LIN {X 0,Y 242.041,Z 125.949,A -85,B 0,C 180,E1 -19236.009,E2 -19236.009} C_VEL
LIN {X 0,Y 242.05,Z 125.947,A -85,B 0,C 180,E1 -19239.604,E2 -19239.604} C_VEL
LIN {X 0,Y 242.178,Z 125.932,A -85,B 0,C 180,E1 -19243.274,E2 -19243.274} C_VEL
LIN {X 0,Y 242.183,Z 125.929,A -85,B 0,C 180,E1 -19248.274,E2 -19248.274} C_VEL
LIN {X 0,Y 242.383,Z 125.908,A -85,B 0,C 180,E1 -19251.659,E2 -19251.659} C_VEL
LIN {X 0,Y 242.244,Z 125.935,A -85,B 0,C 180,E1 -19255.002,E2 -19255.002} C_VEL
LIN {X 0,Y 242.634,Z 125.882,A -85,B 0,C 180,E1 -19258.335,E2 -19258.335} C_VEL
LIN {X 0,Y 242.641,Z 125.873,A -85,B 0,C 180,E1 -19261.654,E2 -19261.654} C_VEL
LIN {X 0,Y 242.413,Z 125.908,A -85,B 0,C 180,E1 -19266.654,E2 -19266.654} C_VEL
LIN {X 0,Y 242.272,Z 125.921,A -85,B 0,C 180,E1 -19270.018,E2 -19270.018} C_VEL
LIN {X 0,Y 242.169,Z 125.946,A -85,B 0,C 180,E1 -19275.134,E2 -19275.134} C_VEL
LIN {X 0,Y 242.074,Z 125.958,A -85,B 0,C 180,E1 -19278.618,E2 -19278.618} C_VEL
LIN {X 0,Y 242.029,Z 126.021,A -85,B 0,C 180,E1 -19282.565,E2 -19282.565} C_VEL
LIN {X 0,Y 242.806,Z 128.403,A -85,B 0,C 180,E1 -19282.995,E2 -19282.995} C_VEL
LIN {X 0,Y 244.693,Z 130.652,A -85,B 0,C 180,E1 -19283.815,E2 -19283.815} C_VEL
LIN {X 0,Y 246.169,Z 131.607,A -85,B 0,C 180,E1 -19284.391,E2 -19284.391} C_VEL
LIN {X 0,Y 247.934,Z 134.724,A -85,B 0,C 180,E1 -19285.156,E2 -19285.156} C_VEL
LIN {X 0,Y 250.263,Z 137.17,A -85,B 0,C 180,E1 -19286.045,E2 -19286.045} C_VEL
LIN {X 0,Y 252.842,Z 140.696,A -85,B 0,C 180,E1 -19287.026,E2 -19287.026} C_VEL
LIN {X 0,Y 254.234,Z 142.51,A -85,B 0,C 180,E1 -19287.534,E2 -19287.534} C_VEL
LIN {X 0,Y 258.183,Z 148.167,A -85,B 0,C 180,E1 -19288.938,E2 -19288.938} C_VEL
LIN {X 0,Y 265.416,Z 159.264,A -85,B 0,C 180,E1 -19291.315,E2 -19291.315} C_VEL
LIN {X 0,Y 272.928,Z 172.626,A -85,B 0,C 180,E1 -19293.606,E2 -19293.606} C_VEL
LIN {X 0,Y 279.601,Z 186.169,A -85,B 0,C 180,E1 -19295.519,E2 -19295.519} C_VEL
LIN {X 0,Y 280.351,Z 187.777,A -85,B 0,C 180,E1 -19295.727,E2 -19295.727} C_VEL
LIN {X 0,Y 276.357,Z 261.18,A -85,B 0,C 180,E1 -19297.607,E2 -19297.607} C_VEL
LIN {X 0,Y 274.792,Z 275.361,A -85,B 0,C 180,E1 -19298.216,E2 -19298.216} C_VEL
LIN {X 0,Y 272.705,Z 288.841,A -85,B 0,C 180,E1 -19299.068,E2 -19299.068} C_VEL
LIN {X 0,Y 270.18,Z 301.704,A -85,B 0,C 180,E1 -19300.169,E2 -19300.169} C_VEL
LIN {X 0,Y 267.285,Z 313.739,A -85,B 0,C 180,E1 -19301.491,E2 -19301.491} C_VEL
LIN {X 0,Y 263.786,Z 325.88,A -85,B 0,C 180,E1 -19303.166,E2 -19303.166} C_VEL
LIN {X 0,Y 260.3,Z 336.639,A -85,B 0,C 180,E1 -19305.032,E2 -19305.032} C_VEL
LIN {X 0,Y 256.62,Z 346.76,A -85,B 0,C 180,E1 -19307.207,E2 -19307.207} C_VEL
LIN {X 0,Y 252.911,Z 356.201,A -85,B 0,C 180,E1 -19309.751,E2 -19309.751} C_VEL
LIN {X 0,Y 249.787,Z 363.635,A -85,B 0,C 180,E1 -19312.266,E2 -19312.266} C_VEL
LIN {X 0,Y 246.665,Z 370.6,A -85,B 0,C 180,E1 -19315.258,E2 -19315.258} C_VEL
LIN {X 0,Y 244.554,Z 375.362,A -85,B 0,C 180,E1 -19317.88,E2 -19317.88} C_VEL
LIN {X 0,Y 242.846,Z 379.053,A -85,B 0,C 180,E1 -19320.526,E2 -19320.526} C_VEL
LIN {X 0,Y 241.181,Z 382.568,A -85,B 0,C 180,E1 -19324.079,E2 -19324.079} C_VEL
LIN {X 0,Y 240.608,Z 383.728,A -85,B 0,C 180,E1 -19325.86,E2 -19325.86} C_VEL
LIN {X 0,Y 239.858,Z 384.91,A -85,B 0,C 180,E1 -19329.412,E2 -19329.412} C_VEL
LIN {X 0,Y 239.521,Z 384.657,A -85,B 0,C 180,E1 -19332.935,E2 -19332.935} C_VEL
LIN {X 0,Y 239.567,Z 382.993,A -85,B 0,C 180,E1 -19336.424,E2 -19336.424} C_VEL
LIN {X 0,Y 239.857,Z 379.919,A -85,B 0,C 180,E1 -19339.872,E2 -19339.872} C_VEL
LIN {X 0,Y 240.373,Z 376.626,A -85,B 0,C 180,E1 -19342.437,E2 -19342.437} C_VEL
LIN {X 0,Y 240.994,Z 372.483,A -85,B 0,C 180,E1 -19344.979,E2 -19344.979} C_VEL
LIN {X 0,Y 241.907,Z 367.319,A -85,B 0,C 180,E1 -19347.5,E2 -19347.5} C_VEL
LIN {X 0,Y 243.405,Z 359.946,A -85,B 0,C 180,E1 -19350.411,E2 -19350.411} C_VEL
LIN {X 0,Y 245.384,Z 350.779,A -85,B 0,C 180,E1 -19353.281,E2 -19353.281} C_VEL
LIN {X 0,Y 247.431,Z 341.232,A -85,B 0,C 180,E1 -19355.692,E2 -19355.692} C_VEL
LIN {X 0,Y 249.463,Z 330.6,A -85,B 0,C 180,E1 -19357.892,E2 -19357.892} C_VEL
LIN {X 0,Y 251.81,Z 318.828,A -85,B 0,C 180,E1 -19359.841,E2 -19359.841} C_VEL
LIN {X 0,Y 254.053,Z 305.76,A -85,B 0,C 180,E1 -19361.567,E2 -19361.567} C_VEL
LIN {X 0,Y 255.854,Z 292.944,A -85,B 0,C 180,E1 -19362.894,E2 -19362.894} C_VEL
LIN {X 0,Y 257.346,Z 279.852,A -85,B 0,C 180,E1 -19363.923,E2 -19363.923} C_VEL
LIN {X 0,Y 258.5,Z 265.758,A -85,B 0,C 180,E1 -19364.714,E2 -19364.714} C_VEL
LIN {X 0,Y 259.312,Z 249.37,A -85,B 0,C 180,E1 -19365.27,E2 -19365.27} C_VEL
LIN {X 0,Y 262.369,Z 171.816,A -85,B 0,C 180,E1 -19367.319,E2 -19367.319} C_VEL
LIN {X 0,Y 253.658,Z 149.318,A -85,B 0,C 180,E1 -19369.1,E2 -19369.1} C_VEL
LIN {X 0,Y 248.74,Z 138.889,A -85,B 0,C 180,E1 -19370.096,E2 -19370.096} C_VEL
LIN {X 0,Y 243.439,Z 129.314,A -85,B 0,C 180,E1 -19371.164,E2 -19371.164} C_VEL
LIN {X 0,Y 242.187,Z 126.552,A -85,B 0,C 180,E1 -19371.442,E2 -19371.442} C_VEL
LIN {X 0,Y 242.072,Z 125.958,A -85,B 0,C 180,E1 -19371.532,E2 -19371.532} C_VEL
LIN {X 0,Y 242.035,Z 125.96,A -85,B 0,C 180,E1 -19375.839,E2 -19375.839} C_VEL
LIN {X 0,Y 241.999,Z 125.965,A -85,B 0,C 180,E1 -19379.581,E2 -19379.581} C_VEL
LIN {X 0,Y 241.961,Z 125.971,A -85,B 0,C 180,E1 -19383.493,E2 -19383.493} C_VEL
LIN {X 0,Y 242.004,Z 125.964,A -85,B 0,C 180,E1 -19387.576,E2 -19387.576} C_VEL
LIN {X 0,Y 242.025,Z 125.957,A -85,B 0,C 180,E1 -19391.9,E2 -19391.9} C_VEL
LIN {X 0,Y 241.997,Z 125.962,A -85,B 0,C 180,E1 -19396.552,E2 -19396.552} C_VEL
LIN {X 0,Y 241.984,Z 125.953,A -85,B 0,C 180,E1 -19400.295,E2 -19400.295} C_VEL
LIN {X 0,Y 242.012,Z 125.957,A -85,B 0,C 180,E1 -19404.501,E2 -19404.501} C_VEL
LIN {X 0,Y 241.951,Z 125.964,A -85,B 0,C 180,E1 -19408.484,E2 -19408.484} C_VEL
LIN {X 0,Y 241.982,Z 125.944,A -85,B 0,C 180,E1 -19412.317,E2 -19412.317} C_VEL
LIN {X 0,Y 242.062,Z 125.957,A -85,B 0,C 180,E1 -19416.023,E2 -19416.023} C_VEL
LIN {X 0,Y 242.068,Z 125.952,A -85,B 0,C 180,E1 -19419.617,E2 -19419.617} C_VEL
LIN {X 0,Y 242.146,Z 125.946,A -85,B 0,C 180,E1 -19423.283,E2 -19423.283} C_VEL
LIN {X 0,Y 242.172,Z 125.942,A -85,B 0,C 180,E1 -19428.285,E2 -19428.285} C_VEL
LIN {X 0,Y 242.421,Z 125.897,A -85,B 0,C 180,E1 -19431.671,E2 -19431.671} C_VEL
LIN {X 0,Y 242.251,Z 125.913,A -85,B 0,C 180,E1 -19435.013,E2 -19435.013} C_VEL
LIN {X 0,Y 242.629,Z 125.884,A -85,B 0,C 180,E1 -19438.346,E2 -19438.346} C_VEL
LIN {X 0,Y 242.628,Z 125.879,A -85,B 0,C 180,E1 -19441.665,E2 -19441.665} C_VEL
LIN {X 0,Y 242.253,Z 125.909,A -85,B 0,C 180,E1 -19444.875,E2 -19444.875} C_VEL
LIN {X 0,Y 241.585,Z 126.003,A -85,B 0,C 180,E1 -19446.265,E2 -19446.265} C_VEL
LIN {X 0,Y 238.754,Z 126.366,A -85,B 0,C 180,E1 -19448.532,E2 -19448.532} C_VEL
LIN {X 0,Y 235.487,Z 126.773,A -85,B 0,C 180,E1 -19451.328,E2 -19451.328} C_VEL
LIN {X 0,Y 235.124,Z 126.815,A -85,B 0,C 180,E1 -19452.297,E2 -19452.297} C_VEL
LIN {X 0,Y 235.092,Z 126.822,A -85,B 0,C 180,E1 -19456.946,E2 -19456.946} C_VEL
LIN {X 0,Y 234.991,Z 126.837,A -85,B 0,C 180,E1 -19462.015,E2 -19462.015} C_VEL
LIN {X 0,Y 234.969,Z 126.835,A -85,B 0,C 180,E1 -19466.663,E2 -19466.663} C_VEL
LIN {X 0,Y 234.932,Z 126.843,A -85,B 0,C 180,E1 -19470.573,E2 -19470.573} C_VEL
LIN {X 0,Y 234.932,Z 126.844,A -85,B 0,C 180,E1 -19474.643,E2 -19474.643} C_VEL
LIN {X 0,Y 234.916,Z 126.844,A -85,B 0,C 180,E1 -19478.941,E2 -19478.941} C_VEL
LIN {X 0,Y 234.882,Z 126.853,A -85,B 0,C 180,E1 -19483.493,E2 -19483.493} C_VEL
LIN {X 0,Y 234.883,Z 126.853,A -85,B 0,C 180,E1 -19486.517,E2 -19486.517} C_VEL
LIN {X 0,Y 234.919,Z 127.017,A -85,B 0,C 180,E1 -19488.637,E2 -19488.637} C_VEL
LIN {X 0,Y 236.99,Z 134.697,A -85,B 0,C 180,E1 -19491.697,E2 -19491.697} C_VEL
LIN {X 0,Y 243.013,Z 147.893,A -85,B 0,C 180,E1 -19493.045,E2 -19493.045} C_VEL
LIN {X 0,Y 251.14,Z 167.812,A -85,B 0,C 180,E1 -19494.814,E2 -19494.814} C_VEL
LIN {X 0,Y 253.217,Z 173.701,A -85,B 0,C 180,E1 -19495.269,E2 -19495.269} C_VEL
LIN {X 0,Y 255.518,Z 191.759,A -85,B 0,C 180,E1 -19496.129,E2 -19496.129} C_VEL
LIN {X 0,Y 252.428,Z 272.237,A -85,B 0,C 180,E1 -19498.359,E2 -19498.359} C_VEL
LIN {X 0,Y 251.193,Z 286.32,A -85,B 0,C 180,E1 -19499.007,E2 -19499.007} C_VEL
LIN {X 0,Y 249.679,Z 299.519,A -85,B 0,C 180,E1 -19499.911,E2 -19499.911} C_VEL
LIN {X 0,Y 247.651,Z 313.005,A -85,B 0,C 180,E1 -19501.158,E2 -19501.158} C_VEL
LIN {X 0,Y 245.502,Z 326.007,A -85,B 0,C 180,E1 -19502.743,E2 -19502.743} C_VEL
LIN {X 0,Y 243.137,Z 337.78,A -85,B 0,C 180,E1 -19504.537,E2 -19504.537} C_VEL
LIN {X 0,Y 241.554,Z 345.588,A -85,B 0,C 180,E1 -19505.966,E2 -19505.966} C_VEL
LIN {X 0,Y 239.418,Z 355.067,A -85,B 0,C 180,E1 -19508.024,E2 -19508.024} C_VEL
LIN {X 0,Y 237.365,Z 364.58,A -85,B 0,C 180,E1 -19510.546,E2 -19510.546} C_VEL
LIN {X 0,Y 235.614,Z 373.622,A -85,B 0,C 180,E1 -19513.541,E2 -19513.541} C_VEL
LIN {X 0,Y 234.356,Z 379.977,A -85,B 0,C 180,E1 -19516.121,E2 -19516.121} C_VEL
LIN {X 0,Y 233.464,Z 385.192,A -85,B 0,C 180,E1 -19518.719,E2 -19518.719} C_VEL
LIN {X 0,Y 233,Z 389.396,A -85,B 0,C 180,E1 -19521.328,E2 -19521.328} C_VEL
LIN {X 0,Y 232.741,Z 393.621,A -85,B 0,C 180,E1 -19524.805,E2 -19524.805} C_VEL
LIN {X 0,Y 232.76,Z 396.365,A -85,B 0,C 180,E1 -19528.272,E2 -19528.272} C_VEL
LIN {X 0,Y 232.83,Z 397.21,A -85,B 0,C 180,E1 -19530.002,E2 -19530.002} C_VEL
LIN {X 0,Y 232.667,Z 397.873,A -85,B 0,C 180,E1 -19533.466,E2 -19533.466} C_VEL
LIN {X 0,Y 232.829,Z 397.211,A -85,B 0,C 180,E1 -19536.937,E2 -19536.937} C_VEL
LIN {X 0,Y 233.482,Z 395.231,A -85,B 0,C 180,E1 -19540.407,E2 -19540.407} C_VEL
LIN {X 0,Y 234.709,Z 391.888,A -85,B 0,C 180,E1 -19543.862,E2 -19543.862} C_VEL
LIN {X 0,Y 236.804,Z 387.097,A -85,B 0,C 180,E1 -19547.267,E2 -19547.267} C_VEL
LIN {X 0,Y 239.552,Z 380.722,A -85,B 0,C 180,E1 -19550.616,E2 -19550.616} C_VEL
LIN {X 0,Y 242.692,Z 373.665,A -85,B 0,C 180,E1 -19553.467,E2 -19553.467} C_VEL
LIN {X 0,Y 245.851,Z 366.318,A -85,B 0,C 180,E1 -19555.848,E2 -19555.848} C_VEL
LIN {X 0,Y 249.475,Z 357.524,A -85,B 0,C 180,E1 -19558.158,E2 -19558.158} C_VEL
LIN {X 0,Y 253.373,Z 347.313,A -85,B 0,C 180,E1 -19560.318,E2 -19560.318} C_VEL
LIN {X 0,Y 256.969,Z 336.685,A -85,B 0,C 180,E1 -19562.14,E2 -19562.14} C_VEL
LIN {X 0,Y 260.744,Z 324.554,A -85,B 0,C 180,E1 -19563.776,E2 -19563.776} C_VEL
LIN {X 0,Y 263.987,Z 311.763,A -85,B 0,C 180,E1 -19565.152,E2 -19565.152} C_VEL
LIN {X 0,Y 266.924,Z 298.45,A -85,B 0,C 180,E1 -19566.214,E2 -19566.214} C_VEL
LIN {X 0,Y 269.32,Z 283.857,A -85,B 0,C 180,E1 -19567.059,E2 -19567.059} C_VEL
LIN {X 0,Y 270.863,Z 269.38,A -85,B 0,C 180,E1 -19567.616,E2 -19567.616} C_VEL
LIN {X 0,Y 274.782,Z 197.77,A -85,B 0,C 180,E1 -19569.471,E2 -19569.471} C_VEL
LIN {X 0,Y 268.635,Z 183.99,A -85,B 0,C 180,E1 -19571.343,E2 -19571.343} C_VEL
LIN {X 0,Y 262.523,Z 172.024,A -85,B 0,C 180,E1 -19573.303,E2 -19573.303} C_VEL
LIN {X 0,Y 257.036,Z 162.531,A -85,B 0,C 180,E1 -19575.163,E2 -19575.163} C_VEL
LIN {X 0,Y 252.081,Z 154.456,A -85,B 0,C 180,E1 -19576.971,E2 -19576.971} C_VEL
LIN {X 0,Y 248.527,Z 149.046,A -85,B 0,C 180,E1 -19578.348,E2 -19578.348} C_VEL
LIN {X 0,Y 244.891,Z 143.679,A -85,B 0,C 180,E1 -19579.843,E2 -19579.843} C_VEL
LIN {X 0,Y 241.577,Z 138.818,A -85,B 0,C 180,E1 -19581.309,E2 -19581.309} C_VEL
LIN {X 0,Y 237.543,Z 133.584,A -85,B 0,C 180,E1 -19583.203,E2 -19583.203} C_VEL
LIN {X 0,Y 236.83,Z 132.267,A -85,B 0,C 180,E1 -19583.588,E2 -19583.588} C_VEL
LIN {X 0,Y 235.994,Z 129.663,A -85,B 0,C 180,E1 -19585.535,E2 -19585.535} C_VEL
LIN {X 0,Y 234.948,Z 126.839,A -85,B 0,C 180,E1 -19587.925,E2 -19587.925} C_VEL
LIN {X 0,Y 234.918,Z 126.842,A -85,B 0,C 180,E1 -19591.396,E2 -19591.396} C_VEL
LIN {X 0,Y 234.97,Z 126.832,A -85,B 0,C 180,E1 -19595.239,E2 -19595.239} C_VEL
LIN {X 0,Y 235.013,Z 126.827,A -85,B 0,C 180,E1 -19598.965,E2 -19598.965} C_VEL
LIN {X 0,Y 235.111,Z 126.814,A -85,B 0,C 180,E1 -19603.056,E2 -19603.056} C_VEL
LIN {X 0,Y 235.116,Z 126.81,A -85,B 0,C 180,E1 -19607.917,E2 -19607.917} C_VEL
LIN {X 0,Y 235.323,Z 126.789,A -85,B 0,C 180,E1 -19611.407,E2 -19611.407} C_VEL
LIN {X 0,Y 235.36,Z 126.78,A -85,B 0,C 180,E1 -19613.135,E2 -19613.135} C_VEL
LIN {X 0,Y 235.593,Z 126.758,A -85,B 0,C 180,E1 -19618.285,E2 -19618.285} C_VEL
LIN {X 0,Y 235.6,Z 126.749,A -85,B 0,C 180,E1 -19621.704,E2 -19621.704} C_VEL
LIN {X 0,Y 235.364,Z 126.788,A -85,B 0,C 180,E1 -19626.854,E2 -19626.854} C_VEL
LIN {X 0,Y 235.219,Z 126.802,A -85,B 0,C 180,E1 -19630.321,E2 -19630.321} C_VEL
LIN {X 0,Y 235.116,Z 126.82,A -85,B 0,C 180,E1 -19635.6,E2 -19635.6} C_VEL
LIN {X 0,Y 234.996,Z 126.84,A -85,B 0,C 180,E1 -19639.711,E2 -19639.711} C_VEL
LIN {X 0,Y 235.78,Z 129.313,A -85,B 0,C 180,E1 -19640.21,E2 -19640.21} C_VEL
LIN {X 0,Y 237.696,Z 131.568,A -85,B 0,C 180,E1 -19641.16,E2 -19641.16} C_VEL
LIN {X 0,Y 239.366,Z 132.759,A -85,B 0,C 180,E1 -19641.909,E2 -19641.909} C_VEL
LIN {X 0,Y 241.227,Z 135.882,A -85,B 0,C 180,E1 -19642.814,E2 -19642.814} C_VEL
LIN {X 0,Y 243.587,Z 138.113,A -85,B 0,C 180,E1 -19643.817,E2 -19643.817} C_VEL
LIN {X 0,Y 245.898,Z 141.51,A -85,B 0,C 180,E1 -19644.814,E2 -19644.814} C_VEL
LIN {X 0,Y 247.465,Z 143.234,A -85,B 0,C 180,E1 -19645.432,E2 -19645.432} C_VEL
LIN {X 0,Y 251.784,Z 149.168,A -85,B 0,C 180,E1 -19647.107,E2 -19647.107} C_VEL
LIN {X 0,Y 254.835,Z 153.563,A -85,B 0,C 180,E1 -19648.228,E2 -19648.228} C_VEL
LIN {X 0,Y 261.686,Z 164.264,A -85,B 0,C 180,E1 -19650.577,E2 -19650.577} C_VEL
LIN {X 0,Y 269.258,Z 178.011,A -85,B 0,C 180,E1 -19652.987,E2 -19652.987} C_VEL
LIN {X 0,Y 275.138,Z 190.241,A -85,B 0,C 180,E1 -19654.746,E2 -19654.746} C_VEL
LIN {X 0,Y 271.184,Z 261.131,A -85,B 0,C 180,E1 -19656.594,E2 -19656.594} C_VEL
LIN {X 0,Y 269.572,Z 275.306,A -85,B 0,C 180,E1 -19657.204,E2 -19657.204} C_VEL
LIN {X 0,Y 267.324,Z 289.177,A -85,B 0,C 180,E1 -19658.085,E2 -19658.085} C_VEL
LIN {X 0,Y 264.919,Z 301.058,A -85,B 0,C 180,E1 -19659.104,E2 -19659.104} C_VEL
LIN {X 0,Y 261.708,Z 313.991,A -85,B 0,C 180,E1 -19660.535,E2 -19660.535} C_VEL
LIN {X 0,Y 258.28,Z 325.511,A -85,B 0,C 180,E1 -19662.138,E2 -19662.138} C_VEL
LIN {X 0,Y 254.461,Z 336.758,A -85,B 0,C 180,E1 -19664.099,E2 -19664.099} C_VEL
LIN {X 0,Y 250.95,Z 346.031,A -85,B 0,C 180,E1 -19666.105,E2 -19666.105} C_VEL
LIN {X 0,Y 247.131,Z 355.357,A -85,B 0,C 180,E1 -19668.606,E2 -19668.606} C_VEL
LIN {X 0,Y 243.936,Z 362.668,A -85,B 0,C 180,E1 -19671.057,E2 -19671.057} C_VEL
LIN {X 0,Y 241.337,Z 368.256,A -85,B 0,C 180,E1 -19673.343,E2 -19673.343} C_VEL
LIN {X 0,Y 238.836,Z 373.518,A -85,B 0,C 180,E1 -19676.004,E2 -19676.004} C_VEL
LIN {X 0,Y 236.823,Z 377.698,A -85,B 0,C 180,E1 -19678.711,E2 -19678.711} C_VEL
LIN {X 0,Y 235.202,Z 380.863,A -85,B 0,C 180,E1 -19681.437,E2 -19681.437} C_VEL
LIN {X 0,Y 233.73,Z 383.725,A -85,B 0,C 180,E1 -19685.102,E2 -19685.102} C_VEL
LIN {X 0,Y 232.848,Z 385.078,A -85,B 0,C 180,E1 -19688.763,E2 -19688.763} C_VEL
LIN {X 0,Y 232.438,Z 384.953,A -85,B 0,C 180,E1 -19692.398,E2 -19692.398} C_VEL
LIN {X 0,Y 232.461,Z 383.408,A -85,B 0,C 180,E1 -19696.001,E2 -19696.001} C_VEL
LIN {X 0,Y 232.714,Z 380.456,A -85,B 0,C 180,E1 -19699.558,E2 -19699.558} C_VEL
LIN {X 0,Y 233.214,Z 377.292,A -85,B 0,C 180,E1 -19702.204,E2 -19702.204} C_VEL
LIN {X 0,Y 233.861,Z 373.229,A -85,B 0,C 180,E1 -19704.825,E2 -19704.825} C_VEL
LIN {X 0,Y 234.763,Z 368.191,A -85,B 0,C 180,E1 -19707.424,E2 -19707.424} C_VEL
LIN {X 0,Y 236.274,Z 360.973,A -85,B 0,C 180,E1 -19710.424,E2 -19710.424} C_VEL
LIN {X 0,Y 237.939,Z 353.421,A -85,B 0,C 180,E1 -19712.96,E2 -19712.96} C_VEL
LIN {X 0,Y 240.041,Z 344.038,A -85,B 0,C 180,E1 -19715.538,E2 -19715.538} C_VEL
LIN {X 0,Y 242.243,Z 333.398,A -85,B 0,C 180,E1 -19717.919,E2 -19717.919} C_VEL
LIN {X 0,Y 244.585,Z 322.217,A -85,B 0,C 180,E1 -19719.925,E2 -19719.925} C_VEL
LIN {X 0,Y 246.849,Z 309.877,A -85,B 0,C 180,E1 -19721.702,E2 -19721.702} C_VEL
LIN {X 0,Y 248.676,Z 298.056,A -85,B 0,C 180,E1 -19723.065,E2 -19723.065} C_VEL
LIN {X 0,Y 250.381,Z 285.154,A -85,B 0,C 180,E1 -19724.215,E2 -19724.215} C_VEL
LIN {X 0,Y 251.769,Z 270.528,A -85,B 0,C 180,E1 -19725.168,E2 -19725.168} C_VEL
LIN {X 0,Y 252.65,Z 255.97,A -85,B 0,C 180,E1 -19725.786,E2 -19725.786} C_VEL
LIN {X 0,Y 256.09,Z 173.861,A -85,B 0,C 180,E1 -19728.003,E2 -19728.003} C_VEL
LIN {X 0,Y 249.273,Z 155.648,A -85,B 0,C 180,E1 -19729.466,E2 -19729.466} C_VEL
LIN {X 0,Y 243.752,Z 143.416,A -85,B 0,C 180,E1 -19730.634,E2 -19730.634} C_VEL
LIN {X 0,Y 236.457,Z 130.343,A -85,B 0,C 180,E1 -19732.171,E2 -19732.171} C_VEL
LIN {X 0,Y 235.107,Z 127.529,A -85,B 0,C 180,E1 -19732.483,E2 -19732.483} C_VEL
LIN {X 0,Y 235.004,Z 126.838,A -85,B 0,C 180,E1 -19732.59,E2 -19732.59} C_VEL
LIN {X 0,Y 234.939,Z 126.84,A -85,B 0,C 180,E1 -19736.658,E2 -19736.658} C_VEL
LIN {X 0,Y 234.901,Z 126.848,A -85,B 0,C 180,E1 -19740.569,E2 -19740.569} C_VEL
LIN {X 0,Y 234.93,Z 126.847,A -85,B 0,C 180,E1 -19744.635,E2 -19744.635} C_VEL
LIN {X 0,Y 234.968,Z 126.84,A -85,B 0,C 180,E1 -19748.964,E2 -19748.964} C_VEL
LIN {X 0,Y 234.971,Z 126.822,A -85,B 0,C 180,E1 -19753.463,E2 -19753.463} C_VEL
LIN {X 0,Y 234.97,Z 126.837,A -85,B 0,C 180,E1 -19756.543,E2 -19756.543} C_VEL
LIN {X 0,Y 234.929,Z 126.825,A -85,B 0,C 180,E1 -19761.09,E2 -19761.09} C_VEL
LIN {X 0,Y 234.936,Z 126.841,A -85,B 0,C 180,E1 -19765.371,E2 -19765.371} C_VEL
LIN {X 0,Y 234.9,Z 126.838,A -85,B 0,C 180,E1 -19769.435,E2 -19769.435} C_VEL
LIN {X 0,Y 234.973,Z 126.828,A -85,B 0,C 180,E1 -19773.799,E2 -19773.799} C_VEL
LIN {X 0,Y 235.032,Z 126.828,A -85,B 0,C 180,E1 -19778.979,E2 -19778.979} C_VEL
LIN {X 0,Y 235.099,Z 126.823,A -85,B 0,C 180,E1 -19783.048,E2 -19783.048} C_VEL
LIN {X 0,Y 235.132,Z 126.821,A -85,B 0,C 180,E1 -19787.929,E2 -19787.929} C_VEL
LIN {X 0,Y 235.376,Z 126.776,A -85,B 0,C 180,E1 -19791.42,E2 -19791.42} C_VEL
LIN {X 0,Y 235.393,Z 126.762,A -85,B 0,C 180,E1 -19793.147,E2 -19793.147} C_VEL
LIN {X 0,Y 235.589,Z 126.761,A -85,B 0,C 180,E1 -19798.296,E2 -19798.296} C_VEL
LIN {X 0,Y 235.587,Z 126.755,A -85,B 0,C 180,E1 -19801.715,E2 -19801.715} C_VEL
LIN {X 0,Y 235.397,Z 126.775,A -85,B 0,C 180,E1 -19806.864,E2 -19806.864} C_VEL
LIN {X 0,Y 235.232,Z 126.807,A -85,B 0,C 180,E1 -19810.332,E2 -19810.332} C_VEL
LIN {X 0,Y 235.124,Z 126.815,A -85,B 0,C 180,E1 -19812.297,E2 -19812.297} C_VEL
LIN {X 0,Y 234.395,Z 126.911,A -85,B 0,C 180,E1 -19813.727,E2 -19813.727} C_VEL
LIN {X 0,Y 231.522,Z 127.272,A -85,B 0,C 180,E1 -19816.061,E2 -19816.061} C_VEL
LIN {X 0,Y 229.099,Z 127.578,A -85,B 0,C 180,E1 -19817.962,E2 -19817.962} C_VEL
LIN {X 0,Y 228.036,Z 127.706,A -85,B 0,C 180,E1 -19819.438,E2 -19819.438} C_VEL
LIN {X 0,Y 227.934,Z 127.716,A -85,B 0,C 180,E1 -19819.939,E2 -19819.939} C_VEL
LIN {X 0,Y 227.912,Z 127.717,A -85,B 0,C 180,E1 -19823.638,E2 -19823.638} C_VEL
LIN {X 0,Y 227.886,Z 127.714,A -85,B 0,C 180,E1 -19827.561,E2 -19827.561} C_VEL
LIN {X 0,Y 227.871,Z 127.72,A -85,B 0,C 180,E1 -19831.628,E2 -19831.628} C_VEL
LIN {X 0,Y 227.883,Z 127.722,A -85,B 0,C 180,E1 -19835.877,E2 -19835.877} C_VEL
LIN {X 0,Y 227.814,Z 127.72,A -85,B 0,C 180,E1 -19840.385,E2 -19840.385} C_VEL
LIN {X 0,Y 227.83,Z 127.732,A -85,B 0,C 180,E1 -19845.2,E2 -19845.2} C_VEL
LIN {X 0,Y 227.832,Z 127.813,A -85,B 0,C 180,E1 -19847.766,E2 -19847.766} C_VEL
LIN {X 0,Y 229.635,Z 134.402,A -85,B 0,C 180,E1 -19850.524,E2 -19850.524} C_VEL
LIN {X 0,Y 236.978,Z 150.066,A -85,B 0,C 180,E1 -19852.242,E2 -19852.242} C_VEL
LIN {X 0,Y 245.172,Z 170.193,A -85,B 0,C 180,E1 -19854.105,E2 -19854.105} C_VEL
LIN {X 0,Y 247.226,Z 176.282,A -85,B 0,C 180,E1 -19854.584,E2 -19854.584} C_VEL
LIN {X 0,Y 249.22,Z 192.924,A -85,B 0,C 180,E1 -19855.391,E2 -19855.391} C_VEL
LIN {X 0,Y 246.007,Z 273.065,A -85,B 0,C 180,E1 -19857.675,E2 -19857.675} C_VEL
LIN {X 0,Y 244.653,Z 287.551,A -85,B 0,C 180,E1 -19858.385,E2 -19858.385} C_VEL
LIN {X 0,Y 243.171,Z 299.816,A -85,B 0,C 180,E1 -19859.259,E2 -19859.259} C_VEL
LIN {X 0,Y 241.043,Z 313.377,A -85,B 0,C 180,E1 -19860.554,E2 -19860.554} C_VEL
LIN {X 0,Y 238.851,Z 326.131,A -85,B 0,C 180,E1 -19862.156,E2 -19862.156} C_VEL
LIN {X 0,Y 236.419,Z 337.854,A -85,B 0,C 180,E1 -19863.997,E2 -19863.997} C_VEL
LIN {X 0,Y 234.516,Z 346.612,A -85,B 0,C 180,E1 -19865.668,E2 -19865.668} C_VEL
LIN {X 0,Y 232.381,Z 355.923,A -85,B 0,C 180,E1 -19867.79,E2 -19867.79} C_VEL
LIN {X 0,Y 230.295,Z 365.244,A -85,B 0,C 180,E1 -19870.388,E2 -19870.388} C_VEL
LIN {X 0,Y 228.705,Z 372.993,A -85,B 0,C 180,E1 -19873.029,E2 -19873.029} C_VEL
LIN {X 0,Y 227.413,Z 379.428,A -85,B 0,C 180,E1 -19875.689,E2 -19875.689} C_VEL
LIN {X 0,Y 226.46,Z 384.688,A -85,B 0,C 180,E1 -19878.365,E2 -19878.365} C_VEL
LIN {X 0,Y 225.951,Z 388.963,A -85,B 0,C 180,E1 -19881.056,E2 -19881.056} C_VEL
LIN {X 0,Y 225.655,Z 393.255,A -85,B 0,C 180,E1 -19884.641,E2 -19884.641} C_VEL
LIN {X 0,Y 225.674,Z 396.062,A -85,B 0,C 180,E1 -19888.218,E2 -19888.218} C_VEL
LIN {X 0,Y 225.742,Z 396.939,A -85,B 0,C 180,E1 -19890.003,E2 -19890.003} C_VEL
LIN {X 0,Y 225.587,Z 397.661,A -85,B 0,C 180,E1 -19893.575,E2 -19893.575} C_VEL
LIN {X 0,Y 225.776,Z 397.063,A -85,B 0,C 180,E1 -19897.155,E2 -19897.155} C_VEL
LIN {X 0,Y 226.477,Z 395.156,A -85,B 0,C 180,E1 -19900.733,E2 -19900.733} C_VEL
LIN {X 0,Y 227.802,Z 391.898,A -85,B 0,C 180,E1 -19904.291,E2 -19904.291} C_VEL
LIN {X 0,Y 230.007,Z 387.182,A -85,B 0,C 180,E1 -19907.794,E2 -19907.794} C_VEL
LIN {X 0,Y 232.893,Z 380.883,A -85,B 0,C 180,E1 -19911.233,E2 -19911.233} C_VEL
LIN {X 0,Y 236.193,Z 373.909,A -85,B 0,C 180,E1 -19914.153,E2 -19914.153} C_VEL
LIN {X 0,Y 240.086,Z 365.308,A -85,B 0,C 180,E1 -19916.986,E2 -19916.986} C_VEL
LIN {X 0,Y 243.965,Z 356.35,A -85,B 0,C 180,E1 -19919.325,E2 -19919.325} C_VEL
LIN {X 0,Y 248.246,Z 345.2,A -85,B 0,C 180,E1 -19921.676,E2 -19921.676} C_VEL
LIN {X 0,Y 251.94,Z 334.873,A -85,B 0,C 180,E1 -19923.386,E2 -19923.386} C_VEL
LIN {X 0,Y 255.732,Z 322.702,A -85,B 0,C 180,E1 -19925.01,E2 -19925.01} C_VEL
LIN {X 0,Y 258.748,Z 311.262,A -85,B 0,C 180,E1 -19926.214,E2 -19926.214} C_VEL
LIN {X 0,Y 261.757,Z 297.862,A -85,B 0,C 180,E1 -19927.288,E2 -19927.288} C_VEL
LIN {X 0,Y 264.129,Z 283.895,A -85,B 0,C 180,E1 -19928.098,E2 -19928.098} C_VEL
LIN {X 0,Y 265.728,Z 269.246,A -85,B 0,C 180,E1 -19928.673,E2 -19928.673} C_VEL
LIN {X 0,Y 269.663,Z 200.044,A -85,B 0,C 180,E1 -19930.489,E2 -19930.489} C_VEL
LIN {X 0,Y 263.068,Z 185.311,A -85,B 0,C 180,E1 -19932.613,E2 -19932.613} C_VEL
LIN {X 0,Y 256.274,Z 172.392,A -85,B 0,C 180,E1 -19934.936,E2 -19934.936} C_VEL
LIN {X 0,Y 250.229,Z 162.097,A -85,B 0,C 180,E1 -19937.173,E2 -19937.173} C_VEL
LIN {X 0,Y 245.627,Z 154.89,A -85,B 0,C 180,E1 -19939.01,E2 -19939.01} C_VEL
LIN {X 0,Y 241.85,Z 149.212,A -85,B 0,C 180,E1 -19940.633,E2 -19940.633} C_VEL
LIN {X 0,Y 238.045,Z 143.731,A -85,B 0,C 180,E1 -19942.4,E2 -19942.4} C_VEL
LIN {X 0,Y 234.636,Z 138.912,A -85,B 0,C 180,E1 -19944.109,E2 -19944.109} C_VEL
LIN {X 0,Y 229.339,Z 131.988,A -85,B 0,C 180,E1 -19947.042,E2 -19947.042} C_VEL
LIN {X 0,Y 227.891,Z 127.722,A -85,B 0,C 180,E1 -19950.935,E2 -19950.935} C_VEL
LIN {X 0,Y 227.918,Z 127.719,A -85,B 0,C 180,E1 -19954.419,E2 -19954.419} C_VEL
LIN {X 0,Y 227.971,Z 127.712,A -85,B 0,C 180,E1 -19958.283,E2 -19958.283} C_VEL
LIN {X 0,Y 228.049,Z 127.696,A -85,B 0,C 180,E1 -19962.822,E2 -19962.822} C_VEL
LIN {X 0,Y 228.075,Z 127.688,A -85,B 0,C 180,E1 -19967.538,E2 -19967.538} C_VEL
LIN {X 0,Y 228.265,Z 127.671,A -85,B 0,C 180,E1 -19971.139,E2 -19971.139} C_VEL
LIN {X 0,Y 228.313,Z 127.657,A -85,B 0,C 180,E1 -19972.922,E2 -19972.922} C_VEL
LIN {X 0,Y 228.551,Z 127.634,A -85,B 0,C 180,E1 -19978.232,E2 -19978.232} C_VEL
LIN {X 0,Y 228.559,Z 127.627,A -85,B 0,C 180,E1 -19981.756,E2 -19981.756} C_VEL
LIN {X 0,Y 228.316,Z 127.669,A -85,B 0,C 180,E1 -19987.067,E2 -19987.067} C_VEL
LIN {X 0,Y 228.15,Z 127.685,A -85,B 0,C 180,E1 -19990.645,E2 -19990.645} C_VEL
LIN {X 0,Y 228.067,Z 127.694,A -85,B 0,C 180,E1 -19994.265,E2 -19994.265} C_VEL
LIN {X 0,Y 228.058,Z 127.73,A -85,B 0,C 180,E1 -19996.407,E2 -19996.407} C_VEL
LIN {X 0,Y 228.837,Z 130.173,A -85,B 0,C 180,E1 -19996.994,E2 -19996.994} C_VEL
LIN {X 0,Y 230.684,Z 132.447,A -85,B 0,C 180,E1 -19998.075,E2 -19998.075} C_VEL
LIN {X 0,Y 232.589,Z 133.731,A -85,B 0,C 180,E1 -19999.063,E2 -19999.063} C_VEL
LIN {X 0,Y 234.163,Z 136.565,A -85,B 0,C 180,E1 -19999.956,E2 -19999.956} C_VEL
LIN {X 0,Y 237.055,Z 139.419,A -85,B 0,C 180,E1 -20001.365,E2 -20001.365} C_VEL
LIN {X 0,Y 239.377,Z 142.714,A -85,B 0,C 180,E1 -20002.487,E2 -20002.487} C_VEL
LIN {X 0,Y 241.041,Z 144.439,A -85,B 0,C 180,E1 -20003.223,E2 -20003.223} C_VEL
LIN {X 0,Y 243.796,Z 148.147,A -85,B 0,C 180,E1 -20004.432,E2 -20004.432} C_VEL
LIN {X 0,Y 248.534,Z 154.561,A -85,B 0,C 180,E1 -20006.349,E2 -20006.349} C_VEL
LIN {X 0,Y 251.64,Z 159.131,A -85,B 0,C 180,E1 -20007.538,E2 -20007.538} C_VEL
LIN {X 0,Y 258.312,Z 169.863,A -85,B 0,C 180,E1 -20009.928,E2 -20009.928} C_VEL
LIN {X 0,Y 264.847,Z 181.902,A -85,B 0,C 180,E1 -20012.103,E2 -20012.103} C_VEL
LIN {X 0,Y 270.126,Z 193.055,A -85,B 0,C 180,E1 -20013.767,E2 -20013.767} C_VEL
LIN {X 0,Y 266.046,Z 261.486,A -85,B 0,C 180,E1 -20015.551,E2 -20015.551} C_VEL
LIN {X 0,Y 264.336,Z 275.952,A -85,B 0,C 180,E1 -20016.186,E2 -20016.186} C_VEL
LIN {X 0,Y 262.045,Z 289.581,A -85,B 0,C 180,E1 -20017.068,E2 -20017.068} C_VEL
LIN {X 0,Y 259.318,Z 302.346,A -85,B 0,C 180,E1 -20018.188,E2 -20018.188} C_VEL
LIN {X 0,Y 255.82,Z 315.669,A -85,B 0,C 180,E1 -20019.712,E2 -20019.712} C_VEL
LIN {X 0,Y 252.079,Z 327.478,A -85,B 0,C 180,E1 -20021.426,E2 -20021.426} C_VEL
LIN {X 0,Y 248.479,Z 337.532,A -85,B 0,C 180,E1 -20023.252,E2 -20023.252} C_VEL
LIN {X 0,Y 244.802,Z 346.738,A -85,B 0,C 180,E1 -20025.299,E2 -20025.299} C_VEL
LIN {X 0,Y 240.845,Z 355.939,A -85,B 0,C 180,E1 -20027.841,E2 -20027.841} C_VEL
LIN {X 0,Y 236.956,Z 364.373,A -85,B 0,C 180,E1 -20030.804,E2 -20030.804} C_VEL
LIN {X 0,Y 233.487,Z 371.261,A -85,B 0,C 180,E1 -20033.937,E2 -20033.937} C_VEL
LIN {X 0,Y 231.036,Z 376.121,A -85,B 0,C 180,E1 -20036.798,E2 -20036.798} C_VEL
LIN {X 0,Y 228.579,Z 380.723,A -85,B 0,C 180,E1 -20040.529,E2 -20040.529} C_VEL
LIN {X 0,Y 226.902,Z 383.713,A -85,B 0,C 180,E1 -20044.299,E2 -20044.299} C_VEL
LIN {X 0,Y 225.86,Z 385.199,A -85,B 0,C 180,E1 -20048.072,E2 -20048.072} C_VEL
LIN {X 0,Y 225.583,Z 385.397,A -85,B 0,C 180,E1 -20049.956,E2 -20049.956} C_VEL
LIN {X 0,Y 225.304,Z 384.71,A -85,B 0,C 180,E1 -20053.693,E2 -20053.693} C_VEL
LIN {X 0,Y 225.344,Z 383.823,A -85,B 0,C 180,E1 -20055.549,E2 -20055.549} C_VEL
LIN {X 0,Y 225.56,Z 380.994,A -85,B 0,C 180,E1 -20059.223,E2 -20059.223} C_VEL
LIN {X 0,Y 226.06,Z 377.938,A -85,B 0,C 180,E1 -20061.955,E2 -20061.955} C_VEL
LIN {X 0,Y 226.732,Z 373.956,A -85,B 0,C 180,E1 -20064.662,E2 -20064.662} C_VEL
LIN {X 0,Y 227.625,Z 369.059,A -85,B 0,C 180,E1 -20067.343,E2 -20067.343} C_VEL
LIN {X 0,Y 229.128,Z 361.997,A -85,B 0,C 180,E1 -20070.437,E2 -20070.437} C_VEL
LIN {X 0,Y 231.144,Z 353.251,A -85,B 0,C 180,E1 -20073.484,E2 -20073.484} C_VEL
LIN {X 0,Y 233.294,Z 344.07,A -85,B 0,C 180,E1 -20076.058,E2 -20076.058} C_VEL
LIN {X 0,Y 235.224,Z 335.015,A -85,B 0,C 180,E1 -20078.156,E2 -20078.156} C_VEL
LIN {X 0,Y 237.344,Z 325.31,A -85,B 0,C 180,E1 -20080.016,E2 -20080.016} C_VEL
LIN {X 0,Y 239.608,Z 313.669,A -85,B 0,C 180,E1 -20081.846,E2 -20081.846} C_VEL
LIN {X 0,Y 241.791,Z 300.876,A -85,B 0,C 180,E1 -20083.444,E2 -20083.444} C_VEL
LIN {X 0,Y 243.67,Z 287.614,A -85,B 0,C 180,E1 -20084.722,E2 -20084.722} C_VEL
LIN {X 0,Y 245.188,Z 273.224,A -85,B 0,C 180,E1 -20085.746,E2 -20085.746} C_VEL
LIN {X 0,Y 246.217,Z 258.729,A -85,B 0,C 180,E1 -20086.423,E2 -20086.423} C_VEL
LIN {X 0,Y 249.818,Z 175.537,A -85,B 0,C 180,E1 -20088.737,E2 -20088.737} C_VEL
LIN {X 0,Y 242.961,Z 157.286,A -85,B 0,C 180,E1 -20090.27,E2 -20090.27} C_VEL
LIN {X 0,Y 238.228,Z 146.914,A -85,B 0,C 180,E1 -20091.312,E2 -20091.312} C_VEL
LIN {X 0,Y 231.277,Z 134.456,A -85,B 0,C 180,E1 -20092.841,E2 -20092.841} C_VEL
LIN {X 0,Y 229.453,Z 131.332,A -85,B 0,C 180,E1 -20093.256,E2 -20093.256} C_VEL
LIN {X 0,Y 228.108,Z 128.691,A -85,B 0,C 180,E1 -20093.581,E2 -20093.581} C_VEL
LIN {X 0,Y 227.923,Z 127.72,A -85,B 0,C 180,E1 -20093.689,E2 -20093.689} C_VEL
LIN {X 0,Y 227.855,Z 127.72,A -85,B 0,C 180,E1 -20097.556,E2 -20097.556} C_VEL
LIN {X 0,Y 227.842,Z 127.729,A -85,B 0,C 180,E1 -20101.623,E2 -20101.623} C_VEL
LIN {X 0,Y 227.889,Z 127.721,A -85,B 0,C 180,E1 -20105.867,E2 -20105.867} C_VEL
LIN {X 0,Y 227.904,Z 127.721,A -85,B 0,C 180,E1 -20110.356,E2 -20110.356} C_VEL
LIN {X 0,Y 227.894,Z 127.707,A -85,B 0,C 180,E1 -20114.833,E2 -20114.833} C_VEL
LIN {X 0,Y 227.908,Z 127.718,A -85,B 0,C 180,E1 -20117.735,E2 -20117.735} C_VEL
LIN {X 0,Y 227.846,Z 127.703,A -85,B 0,C 180,E1 -20121.918,E2 -20121.918} C_VEL
LIN {X 0,Y 227.867,Z 127.725,A -85,B 0,C 180,E1 -20126.377,E2 -20126.377} C_VEL
LIN {X 0,Y 227.882,Z 127.699,A -85,B 0,C 180,E1 -20130.44,E2 -20130.44} C_VEL
LIN {X 0,Y 227.913,Z 127.711,A -85,B 0,C 180,E1 -20134.431,E2 -20134.431} C_VEL
LIN {X 0,Y 227.992,Z 127.707,A -85,B 0,C 180,E1 -20138.297,E2 -20138.297} C_VEL
LIN {X 0,Y 228.028,Z 127.704,A -85,B 0,C 180,E1 -20142.822,E2 -20142.822} C_VEL
LIN {X 0,Y 228.079,Z 127.698,A -85,B 0,C 180,E1 -20147.55,E2 -20147.55} C_VEL
LIN {X 0,Y 228.311,Z 127.658,A -85,B 0,C 180,E1 -20151.152,E2 -20151.152} C_VEL
LIN {X 0,Y 228.345,Z 127.639,A -85,B 0,C 180,E1 -20152.934,E2 -20152.934} C_VEL
LIN {X 0,Y 228.547,Z 127.638,A -85,B 0,C 180,E1 -20158.244,E2 -20158.244} C_VEL
LIN {X 0,Y 228.546,Z 127.631,A -85,B 0,C 180,E1 -20161.768,E2 -20161.768} C_VEL
LIN {X 0,Y 228.348,Z 127.654,A -85,B 0,C 180,E1 -20167.077,E2 -20167.077} C_VEL
LIN {X 0,Y 228.157,Z 127.69,A -85,B 0,C 180,E1 -20170.656,E2 -20170.656} C_VEL
LIN {X 0,Y 228.06,Z 127.7,A -85,B 0,C 180,E1 -20174.278,E2 -20174.278} C_VEL
LIN {X 0,Y 228,Z 127.705,A -85,B 0,C 180,E1 -20177.959,E2 -20177.959} C_VEL
LIN {X 0,Y 227.934,Z 127.716,A -85,B 0,C 180,E1 -20179.939,E2 -20179.939} C_VEL
LIN {X 0,Y 227.23,Z 127.804,A -85,B 0,C 180,E1 -20181.413,E2 -20181.413} C_VEL
LIN {X 0,Y 224.384,Z 128.157,A -85,B 0,C 180,E1 -20183.819,E2 -20183.819} C_VEL
LIN {X 0,Y 221.978,Z 128.457,A -85,B 0,C 180,E1 -20185.782,E2 -20185.782} C_VEL
LIN {X 0,Y 220.934,Z 128.58,A -85,B 0,C 180,E1 -20187.305,E2 -20187.305} C_VEL
LIN {X 0,Y 220.841,Z 128.59,A -85,B 0,C 180,E1 -20187.822,E2 -20187.822} C_VEL
LIN {X 0,Y 220.839,Z 128.597,A -85,B 0,C 180,E1 -20190.773,E2 -20190.773} C_VEL
LIN {X 0,Y 220.803,Z 128.603,A -85,B 0,C 180,E1 -20194.96,E2 -20194.96} C_VEL
LIN {X 0,Y 220.812,Z 128.603,A -85,B 0,C 180,E1 -20197.284,E2 -20197.284} C_VEL
LIN {X 0,Y 220.766,Z 128.606,A -85,B 0,C 180,E1 -20201.96,E2 -20201.96} C_VEL
LIN {X 0,Y 220.762,Z 128.612,A -85,B 0,C 180,E1 -20206.655,E2 -20206.655} C_VEL
LIN {X 0,Y 220.856,Z 129.102,A -85,B 0,C 180,E1 -20207.052,E2 -20207.052} C_VEL
LIN {X 0,Y 222.259,Z 134.187,A -85,B 0,C 180,E1 -20209.256,E2 -20209.256} C_VEL
LIN {X 0,Y 230.021,Z 150.129,A -85,B 0,C 180,E1 -20211.172,E2 -20211.172} C_VEL
LIN {X 0,Y 238.229,Z 170.034,A -85,B 0,C 180,E1 -20213.129,E2 -20213.129} C_VEL
LIN {X 0,Y 241.229,Z 178.552,A -85,B 0,C 180,E1 -20213.85,E2 -20213.85} C_VEL
LIN {X 0,Y 243.009,Z 193.245,A -85,B 0,C 180,E1 -20214.594,E2 -20214.594} C_VEL
LIN {X 0,Y 239.705,Z 272.653,A -85,B 0,C 180,E1 -20216.905,E2 -20216.905} C_VEL
LIN {X 0,Y 238.32,Z 287.215,A -85,B 0,C 180,E1 -20217.631,E2 -20217.631} C_VEL
LIN {X 0,Y 236.696,Z 300.084,A -85,B 0,C 180,E1 -20218.572,E2 -20218.572} C_VEL
LIN {X 0,Y 234.54,Z 313.367,A -85,B 0,C 180,E1 -20219.876,E2 -20219.876} C_VEL
LIN {X 0,Y 232.375,Z 325.522,A -85,B 0,C 180,E1 -20221.435,E2 -20221.435} C_VEL
LIN {X 0,Y 229.721,Z 337.901,A -85,B 0,C 180,E1 -20223.424,E2 -20223.424} C_VEL
LIN {X 0,Y 228.045,Z 345.635,A -85,B 0,C 180,E1 -20224.931,E2 -20224.931} C_VEL
LIN {X 0,Y 225.737,Z 355.061,A -85,B 0,C 180,E1 -20227.1,E2 -20227.1} C_VEL
LIN {X 0,Y 223.528,Z 364.498,A -85,B 0,C 180,E1 -20229.769,E2 -20229.769} C_VEL
LIN {X 0,Y 221.77,Z 372.454,A -85,B 0,C 180,E1 -20232.528,E2 -20232.528} C_VEL
LIN {X 0,Y 220.49,Z 378.838,A -85,B 0,C 180,E1 -20235.229,E2 -20235.229} C_VEL
LIN {X 0,Y 219.445,Z 384.17,A -85,B 0,C 180,E1 -20237.988,E2 -20237.988} C_VEL
LIN {X 0,Y 218.777,Z 389.78,A -85,B 0,C 180,E1 -20241.691,E2 -20241.691} C_VEL
LIN {X 0,Y 218.527,Z 393.934,A -85,B 0,C 180,E1 -20245.6,E2 -20245.6} C_VEL
LIN {X 0,Y 218.571,Z 395.756,A -85,B 0,C 180,E1 -20248.16,E2 -20248.16} C_VEL
LIN {X 0,Y 218.656,Z 396.664,A -85,B 0,C 180,E1 -20250.003,E2 -20250.003} C_VEL
LIN {X 0,Y 218.514,Z 397.449,A -85,B 0,C 180,E1 -20253.691,E2 -20253.691} C_VEL
LIN {X 0,Y 218.697,Z 396.913,A -85,B 0,C 180,E1 -20257.388,E2 -20257.388} C_VEL
LIN {X 0,Y 219.45,Z 395.07,A -85,B 0,C 180,E1 -20261.081,E2 -20261.081} C_VEL
LIN {X 0,Y 220.912,Z 391.888,A -85,B 0,C 180,E1 -20264.747,E2 -20264.747} C_VEL
LIN {X 0,Y 223.236,Z 387.266,A -85,B 0,C 180,E1 -20268.353,E2 -20268.353} C_VEL
LIN {X 0,Y 226.256,Z 381.044,A -85,B 0,C 180,E1 -20271.888,E2 -20271.888} C_VEL
LIN {X 0,Y 229.709,Z 374.161,A -85,B 0,C 180,E1 -20274.88,E2 -20274.88} C_VEL
LIN {X 0,Y 233.781,Z 365.665,A -85,B 0,C 180,E1 -20277.775,E2 -20277.775} C_VEL
LIN {X 0,Y 237.829,Z 356.824,A -85,B 0,C 180,E1 -20280.159,E2 -20280.159} C_VEL
LIN {X 0,Y 242.177,Z 346.013,A -85,B 0,C 180,E1 -20282.514,E2 -20282.514} C_VEL
LIN {X 0,Y 246.081,Z 335.642,A -85,B 0,C 180,E1 -20284.29,E2 -20284.29} C_VEL
LIN {X 0,Y 250.011,Z 323.675,A -85,B 0,C 180,E1 -20285.934,E2 -20285.934} C_VEL
LIN {X 0,Y 253.582,Z 310.765,A -85,B 0,C 180,E1 -20287.322,E2 -20287.322} C_VEL
LIN {X 0,Y 256.705,Z 297.247,A -85,B 0,C 180,E1 -20288.401,E2 -20288.401} C_VEL
LIN {X 0,Y 259.151,Z 283.079,A -85,B 0,C 180,E1 -20289.217,E2 -20289.217} C_VEL
LIN {X 0,Y 260.688,Z 269.497,A -85,B 0,C 180,E1 -20289.753,E2 -20289.753} C_VEL
LIN {X 0,Y 264.668,Z 202.621,A -85,B 0,C 180,E1 -20291.524,E2 -20291.524} C_VEL
LIN {X 0,Y 258.89,Z 189.509,A -85,B 0,C 180,E1 -20293.493,E2 -20293.493} C_VEL
LIN {X 0,Y 252.389,Z 176.857,A -85,B 0,C 180,E1 -20295.83,E2 -20295.83} C_VEL
LIN {X 0,Y 246.051,Z 165.915,A -85,B 0,C 180,E1 -20298.311,E2 -20298.311} C_VEL
LIN {X 0,Y 239.482,Z 155.543,A -85,B 0,C 180,E1 -20301.166,E2 -20301.166} C_VEL
LIN {X 0,Y 235.345,Z 149.583,A -85,B 0,C 180,E1 -20303.155,E2 -20303.155} C_VEL
LIN {X 0,Y 231.399,Z 143.986,A -85,B 0,C 180,E1 -20305.237,E2 -20305.237} C_VEL
LIN {X 0,Y 226.622,Z 137.635,A -85,B 0,C 180,E1 -20308.047,E2 -20308.047} C_VEL
LIN {X 0,Y 223.125,Z 133.551,A -85,B 0,C 180,E1 -20310.382,E2 -20310.382} C_VEL
LIN {X 0,Y 221.758,Z 131.261,A -85,B 0,C 180,E1 -20311.481,E2 -20311.481} C_VEL
LIN {X 0,Y 220.876,Z 128.594,A -85,B 0,C 180,E1 -20314.555,E2 -20314.555} C_VEL
LIN {X 0,Y 220.902,Z 128.581,A -85,B 0,C 180,E1 -20319.509,E2 -20319.509} C_VEL
LIN {X 0,Y 221.029,Z 128.565,A -85,B 0,C 180,E1 -20323.366,E2 -20323.366} C_VEL
LIN {X 0,Y 221.077,Z 128.56,A -85,B 0,C 180,E1 -20328.998,E2 -20328.998} C_VEL
LIN {X 0,Y 221.251,Z 128.536,A -85,B 0,C 180,E1 -20332.695,E2 -20332.695} C_VEL
LIN {X 0,Y 221.484,Z 128.513,A -85,B 0,C 180,E1 -20338.176,E2 -20338.176} C_VEL
LIN {X 0,Y 221.517,Z 128.504,A -85,B 0,C 180,E1 -20341.812,E2 -20341.812} C_VEL
LIN {X 0,Y 221.253,Z 128.551,A -85,B 0,C 180,E1 -20347.293,E2 -20347.293} C_VEL
LIN {X 0,Y 221.086,Z 128.568,A -85,B 0,C 180,E1 -20350.989,E2 -20350.989} C_VEL
LIN {X 0,Y 221.044,Z 128.606,A -85,B 0,C 180,E1 -20352.27,E2 -20352.27} C_VEL
LIN {X 0,Y 221.731,Z 130.87,A -85,B 0,C 180,E1 -20352.929,E2 -20352.929} C_VEL
LIN {X 0,Y 223.318,Z 132.979,A -85,B 0,C 180,E1 -20354.11,E2 -20354.11} C_VEL
LIN {X 0,Y 225.876,Z 134.608,A -85,B 0,C 180,E1 -20355.734,E2 -20355.734} C_VEL
LIN {X 0,Y 227.463,Z 137.602,A -85,B 0,C 180,E1 -20356.815,E2 -20356.815} C_VEL
LIN {X 0,Y 229.81,Z 139.749,A -85,B 0,C 180,E1 -20358.146,E2 -20358.146} C_VEL
LIN {X 0,Y 230.511,Z 140.614,A -85,B 0,C 180,E1 -20358.542,E2 -20358.542} C_VEL
LIN {X 0,Y 232.911,Z 143.956,A -85,B 0,C 180,E1 -20359.866,E2 -20359.866} C_VEL
LIN {X 0,Y 234.567,Z 145.528,A -85,B 0,C 180,E1 -20360.688,E2 -20360.688} C_VEL
LIN {X 0,Y 237.21,Z 149.175,A -85,B 0,C 180,E1 -20362.003,E2 -20362.003} C_VEL
LIN {X 0,Y 238.779,Z 151.05,A -85,B 0,C 180,E1 -20362.731,E2 -20362.731} C_VEL
LIN {X 0,Y 242.458,Z 156.028,A -85,B 0,C 180,E1 -20364.376,E2 -20364.376} C_VEL
LIN {X 0,Y 247.469,Z 162.933,A -85,B 0,C 180,E1 -20366.421,E2 -20366.421} C_VEL
LIN {X 0,Y 254.727,Z 175.017,A -85,B 0,C 180,E1 -20369.174,E2 -20369.174} C_VEL
LIN {X 0,Y 260.825,Z 186.454,A -85,B 0,C 180,E1 -20371.294,E2 -20371.294} C_VEL
LIN {X 0,Y 265.083,Z 195.475,A -85,B 0,C 180,E1 -20372.709,E2 -20372.709} C_VEL
LIN {X 0,Y 260.989,Z 262.112,A -85,B 0,C 180,E1 -20374.482,E2 -20374.482} C_VEL
LIN {X 0,Y 259.185,Z 276.585,A -85,B 0,C 180,E1 -20375.127,E2 -20375.127} C_VEL
LIN {X 0,Y 256.839,Z 289.974,A -85,B 0,C 180,E1 -20376.005,E2 -20376.005} C_VEL
LIN {X 0,Y 254.051,Z 302.611,A -85,B 0,C 180,E1 -20377.13,E2 -20377.13} C_VEL
LIN {X 0,Y 250.625,Z 315.24,A -85,B 0,C 180,E1 -20378.583,E2 -20378.583} C_VEL
LIN {X 0,Y 247.053,Z 326.081,A -85,B 0,C 180,E1 -20380.133,E2 -20380.133} C_VEL
LIN {X 0,Y 242.944,Z 337.292,A -85,B 0,C 180,E1 -20382.155,E2 -20382.155} C_VEL
LIN {X 0,Y 238.74,Z 347.431,A -85,B 0,C 180,E1 -20384.446,E2 -20384.446} C_VEL
LIN {X 0,Y 234.606,Z 356.542,A -85,B 0,C 180,E1 -20387.035,E2 -20387.035} C_VEL
LIN {X 0,Y 231.328,Z 363.239,A -85,B 0,C 180,E1 -20389.411,E2 -20389.411} C_VEL
LIN {X 0,Y 228.254,Z 369.165,A -85,B 0,C 180,E1 -20391.987,E2 -20391.987} C_VEL
LIN {X 0,Y 225.482,Z 374.314,A -85,B 0,C 180,E1 -20394.784,E2 -20394.784} C_VEL
LIN {X 0,Y 222.706,Z 379.327,A -85,B 0,C 180,E1 -20398.42,E2 -20398.42} C_VEL
LIN {X 0,Y 220.938,Z 382.337,A -85,B 0,C 180,E1 -20401.498,E2 -20401.498} C_VEL
LIN {X 0,Y 219.402,Z 384.691,A -85,B 0,C 180,E1 -20405.388,E2 -20405.388} C_VEL
LIN {X 0,Y 218.597,Z 385.569,A -85,B 0,C 180,E1 -20409.286,E2 -20409.286} C_VEL
LIN {X 0,Y 218.205,Z 385.019,A -85,B 0,C 180,E1 -20413.147,E2 -20413.147} C_VEL
LIN {X 0,Y 218.247,Z 384.212,A -85,B 0,C 180,E1 -20415.069,E2 -20415.069} C_VEL
LIN {X 0,Y 218.413,Z 381.524,A -85,B 0,C 180,E1 -20418.866,E2 -20418.866} C_VEL
LIN {X 0,Y 219.112,Z 377.342,A -85,B 0,C 180,E1 -20422.626,E2 -20422.626} C_VEL
LIN {X 0,Y 219.808,Z 373.227,A -85,B 0,C 180,E1 -20425.413,E2 -20425.413} C_VEL
LIN {X 0,Y 220.825,Z 368.088,A -85,B 0,C 180,E1 -20428.174,E2 -20428.174} C_VEL
LIN {X 0,Y 222.484,Z 360.757,A -85,B 0,C 180,E1 -20431.355,E2 -20431.355} C_VEL
LIN {X 0,Y 224.357,Z 353.067,A -85,B 0,C 180,E1 -20434.039,E2 -20434.039} C_VEL
LIN {X 0,Y 226.683,Z 343.516,A -85,B 0,C 180,E1 -20436.763,E2 -20436.763} C_VEL
LIN {X 0,Y 229.031,Z 332.668,A -85,B 0,C 180,E1 -20439.268,E2 -20439.268} C_VEL
LIN {X 0,Y 231.618,Z 321.193,A -85,B 0,C 180,E1 -20441.372,E2 -20441.372} C_VEL
LIN {X 0,Y 234.081,Z 308.515,A -85,B 0,C 180,E1 -20443.232,E2 -20443.232} C_VEL
LIN {X 0,Y 236.082,Z 296.236,A -85,B 0,C 180,E1 -20444.655,E2 -20444.655} C_VEL
LIN {X 0,Y 237.859,Z 282.691,A -85,B 0,C 180,E1 -20445.859,E2 -20445.859} C_VEL
LIN {X 0,Y 239.214,Z 268.725,A -85,B 0,C 180,E1 -20446.753,E2 -20446.753} C_VEL
LIN {X 0,Y 240.128,Z 254.019,A -85,B 0,C 180,E1 -20447.353,E2 -20447.353} C_VEL
LIN {X 0,Y 243.604,Z 177.607,A -85,B 0,C 180,E1 -20449.488,E2 -20449.488} C_VEL
LIN {X 0,Y 242.471,Z 173.846,A -85,B 0,C 180,E1 -20449.771,E2 -20449.771} C_VEL
LIN {X 0,Y 235.938,Z 157.181,A -85,B 0,C 180,E1 -20451.289,E2 -20451.289} C_VEL
LIN {X 0,Y 231.476,Z 147.965,A -85,B 0,C 180,E1 -20452.31,E2 -20452.31} C_VEL
LIN {X 0,Y 224.53,Z 135.768,A -85,B 0,C 180,E1 -20453.919,E2 -20453.919} C_VEL
LIN {X 0,Y 222.05,Z 131.682,A -85,B 0,C 180,E1 -20454.512,E2 -20454.512} C_VEL
LIN {X 0,Y 220.907,Z 128.849,A -85,B 0,C 180,E1 -20454.828,E2 -20454.828} C_VEL
LIN {X 0,Y 220.875,Z 128.596,A -85,B 0,C 180,E1 -20454.933,E2 -20454.933} C_VEL
LIN {X 0,Y 220.806,Z 128.602,A -85,B 0,C 180,E1 -20458.515,E2 -20458.515} C_VEL
LIN {X 0,Y 220.794,Z 128.606,A -85,B 0,C 180,E1 -20462.757,E2 -20462.757} C_VEL
LIN {X 0,Y 220.839,Z 128.601,A -85,B 0,C 180,E1 -20467.3,E2 -20467.3} C_VEL
LIN {X 0,Y 220.859,Z 128.592,A -85,B 0,C 180,E1 -20471.928,E2 -20471.928} C_VEL
LIN {X 0,Y 220.848,Z 128.592,A -85,B 0,C 180,E1 -20475.575,E2 -20475.575} C_VEL
LIN {X 0,Y 220.835,Z 128.59,A -85,B 0,C 180,E1 -20479.795,E2 -20479.795} C_VEL
LIN {X 0,Y 220.809,Z 128.582,A -85,B 0,C 180,E1 -20482.799,E2 -20482.799} C_VEL
LIN {X 0,Y 220.8,Z 128.602,A -85,B 0,C 180,E1 -20487.249,E2 -20487.249} C_VEL
LIN {X 0,Y 220.805,Z 128.575,A -85,B 0,C 180,E1 -20491.49,E2 -20491.49} C_VEL
LIN {X 0,Y 220.863,Z 128.595,A -85,B 0,C 180,E1 -20495.572,E2 -20495.572} C_VEL
LIN {X 0,Y 220.908,Z 128.586,A -85,B 0,C 180,E1 -20499.523,E2 -20499.523} C_VEL
LIN {X 0,Y 221.008,Z 128.58,A -85,B 0,C 180,E1 -20503.376,E2 -20503.376} C_VEL
LIN {X 0,Y 221.102,Z 128.566,A -85,B 0,C 180,E1 -20509.012,E2 -20509.012} C_VEL
LIN {X 0,Y 221.282,Z 128.519,A -85,B 0,C 180,E1 -20512.708,E2 -20512.708} C_VEL
LIN {X 0,Y 221.505,Z 128.515,A -85,B 0,C 180,E1 -20518.188,E2 -20518.188} C_VEL
LIN {X 0,Y 221.504,Z 128.508,A -85,B 0,C 180,E1 -20521.824,E2 -20521.824} C_VEL
LIN {X 0,Y 221.283,Z 128.535,A -85,B 0,C 180,E1 -20527.304,E2 -20527.304} C_VEL
LIN {X 0,Y 221.106,Z 128.566,A -85,B 0,C 180,E1 -20531,E2 -20531} C_VEL
LIN {X 0,Y 221.012,Z 128.576,A -85,B 0,C 180,E1 -20536.636,E2 -20536.636} C_VEL
LIN {X 0,Y 220.89,Z 128.595,A -85,B 0,C 180,E1 -20540.492,E2 -20540.492} C_VEL
LIN {X 0,Y 220.866,Z 128.596,A -85,B 0,C 180,E1 -20544.441,E2 -20544.441} C_VEL
LIN {X 0,Y 220.841,Z 128.59,A -85,B 0,C 180,E1 -20547.822,E2 -20547.822} C_VEL
LIN {X 0,Y 220.142,Z 128.684,A -85,B 0,C 180,E1 -20549.342,E2 -20549.342} C_VEL
LIN {X 0,Y 217.262,Z 129.04,A -85,B 0,C 180,E1 -20551.823,E2 -20551.823} C_VEL
LIN {X 0,Y 214.838,Z 129.346,A -85,B 0,C 180,E1 -20553.849,E2 -20553.849} C_VEL
LIN {X 0,Y 213.814,Z 129.473,A -85,B 0,C 180,E1 -20555.423,E2 -20555.423} C_VEL
LIN {X 0,Y 213.739,Z 129.484,A -85,B 0,C 180,E1 -20555.957,E2 -20555.957} C_VEL
LIN {X 0,Y 213.712,Z 129.476,A -85,B 0,C 180,E1 -20560.86,E2 -20560.86} C_VEL
LIN {X 0,Y 213.737,Z 129.594,A -85,B 0,C 180,E1 -20565.917,E2 -20565.917} C_VEL
LIN {X 0,Y 214.817,Z 133.667,A -85,B 0,C 180,E1 -20567.842,E2 -20567.842} C_VEL
LIN {X 0,Y 223.307,Z 150.729,A -85,B 0,C 180,E1 -20570.082,E2 -20570.082} C_VEL
LIN {X 0,Y 230.73,Z 168.416,A -85,B 0,C 180,E1 -20571.956,E2 -20571.956} C_VEL
LIN {X 0,Y 235.202,Z 180.437,A -85,B 0,C 180,E1 -20573.06,E2 -20573.06} C_VEL
LIN {X 0,Y 236.824,Z 194.352,A -85,B 0,C 180,E1 -20573.782,E2 -20573.782} C_VEL
LIN {X 0,Y 233.414,Z 272.217,A -85,B 0,C 180,E1 -20576.088,E2 -20576.088} C_VEL
LIN {X 0,Y 232.038,Z 286.882,A -85,B 0,C 180,E1 -20576.836,E2 -20576.836} C_VEL
LIN {X 0,Y 230.417,Z 299.206,A -85,B 0,C 180,E1 -20577.742,E2 -20577.742} C_VEL
LIN {X 0,Y 228.396,Z 311.756,A -85,B 0,C 180,E1 -20578.978,E2 -20578.978} C_VEL
LIN {X 0,Y 226.066,Z 324.168,A -85,B 0,C 180,E1 -20580.561,E2 -20580.561} C_VEL
LIN {X 0,Y 223.539,Z 335.553,A -85,B 0,C 180,E1 -20582.375,E2 -20582.375} C_VEL
LIN {X 0,Y 221.621,Z 344.635,A -85,B 0,C 180,E1 -20584.152,E2 -20584.152} C_VEL
LIN {X 0,Y 219.134,Z 354.155,A -85,B 0,C 180,E1 -20586.369,E2 -20586.369} C_VEL
LIN {X 0,Y 216.797,Z 363.739,A -85,B 0,C 180,E1 -20589.112,E2 -20589.112} C_VEL
LIN {X 0,Y 214.78,Z 372.436,A -85,B 0,C 180,E1 -20592.214,E2 -20592.214} C_VEL
LIN {X 0,Y 213.157,Z 380.155,A -85,B 0,C 180,E1 -20595.686,E2 -20595.686} C_VEL
LIN {X 0,Y 212.216,Z 385.257,A -85,B 0,C 180,E1 -20598.542,E2 -20598.542} C_VEL
LIN {X 0,Y 211.604,Z 390.487,A -85,B 0,C 180,E1 -20602.368,E2 -20602.368} C_VEL
LIN {X 0,Y 211.434,Z 393.83,A -85,B 0,C 180,E1 -20605.762,E2 -20605.762} C_VEL
LIN {X 0,Y 211.47,Z 395.448,A -85,B 0,C 180,E1 -20608.098,E2 -20608.098} C_VEL
LIN {X 0,Y 211.571,Z 396.389,A -85,B 0,C 180,E1 -20610.003,E2 -20610.003} C_VEL
LIN {X 0,Y 211.413,Z 397.236,A -85,B 0,C 180,E1 -20613.815,E2 -20613.815} C_VEL
LIN {X 0,Y 211.637,Z 396.763,A -85,B 0,C 180,E1 -20617.636,E2 -20617.636} C_VEL
LIN {X 0,Y 212.437,Z 394.984,A -85,B 0,C 180,E1 -20621.452,E2 -20621.452} C_VEL
LIN {X 0,Y 214.036,Z 391.869,A -85,B 0,C 180,E1 -20625.232,E2 -20625.232} C_VEL
LIN {X 0,Y 216.488,Z 387.339,A -85,B 0,C 180,E1 -20628.946,E2 -20628.946} C_VEL
LIN {X 0,Y 219.655,Z 381.223,A -85,B 0,C 180,E1 -20632.581,E2 -20632.581} C_VEL
LIN {X 0,Y 223.264,Z 374.427,A -85,B 0,C 180,E1 -20635.65,E2 -20635.65} C_VEL
LIN {X 0,Y 227.531,Z 366.028,A -85,B 0,C 180,E1 -20638.607,E2 -20638.607} C_VEL
LIN {X 0,Y 231.751,Z 357.298,A -85,B 0,C 180,E1 -20641.036,E2 -20641.036} C_VEL
LIN {X 0,Y 236.174,Z 346.8,A -85,B 0,C 180,E1 -20643.4,E2 -20643.4} C_VEL
LIN {X 0,Y 240.391,Z 336.175,A -85,B 0,C 180,E1 -20645.271,E2 -20645.271} C_VEL
LIN {X 0,Y 244.358,Z 324.646,A -85,B 0,C 180,E1 -20646.9,E2 -20646.9} C_VEL
LIN {X 0,Y 248.025,Z 312.019,A -85,B 0,C 180,E1 -20648.308,E2 -20648.308} C_VEL
LIN {X 0,Y 251.242,Z 298.955,A -85,B 0,C 180,E1 -20649.396,E2 -20649.396} C_VEL
LIN {X 0,Y 253.901,Z 284.888,A -85,B 0,C 180,E1 -20650.255,E2 -20650.255} C_VEL
LIN {X 0,Y 255.63,Z 271.214,A -85,B 0,C 180,E1 -20650.832,E2 -20650.832} C_VEL
LIN {X 0,Y 259.764,Z 205.118,A -85,B 0,C 180,E1 -20652.612,E2 -20652.612} C_VEL
LIN {X 0,Y 254.189,Z 192.428,A -85,B 0,C 180,E1 -20654.618,E2 -20654.618} C_VEL
LIN {X 0,Y 248.172,Z 180.653,A -85,B 0,C 180,E1 -20656.913,E2 -20656.913} C_VEL
LIN {X 0,Y 242.484,Z 170.749,A -85,B 0,C 180,E1 -20659.258,E2 -20659.258} C_VEL
LIN {X 0,Y 238.676,Z 164.578,A -85,B 0,C 180,E1 -20660.966,E2 -20660.966} C_VEL
LIN {X 0,Y 236.095,Z 160.469,A -85,B 0,C 180,E1 -20662.203,E2 -20662.203} C_VEL
LIN {X 0,Y 232.796,Z 155.5,A -85,B 0,C 180,E1 -20663.878,E2 -20663.878} C_VEL
LIN {X 0,Y 229.023,Z 150.09,A -85,B 0,C 180,E1 -20665.954,E2 -20665.954} C_VEL
LIN {X 0,Y 224.465,Z 143.878,A -85,B 0,C 180,E1 -20668.762,E2 -20668.762} C_VEL
LIN {X 0,Y 221.099,Z 139.71,A -85,B 0,C 180,E1 -20671.128,E2 -20671.128} C_VEL
LIN {X 0,Y 219.777,Z 137.705,A -85,B 0,C 180,E1 -20672.182,E2 -20672.182} C_VEL
LIN {X 0,Y 216.445,Z 134.114,A -85,B 0,C 180,E1 -20675.026,E2 -20675.026} C_VEL
LIN {X 0,Y 214.629,Z 131.976,A -85,B 0,C 180,E1 -20676.857,E2 -20676.857} C_VEL
LIN {X 0,Y 214.058,Z 130.555,A -85,B 0,C 180,E1 -20677.661,E2 -20677.661} C_VEL
LIN {X 0,Y 213.852,Z 129.46,A -85,B 0,C 180,E1 -20679.306,E2 -20679.306} C_VEL
LIN {X 0,Y 213.958,Z 129.45,A -85,B 0,C 180,E1 -20682.799,E2 -20682.799} C_VEL
LIN {X 0,Y 213.958,Z 129.454,A -85,B 0,C 180,E1 -20686.701,E2 -20686.701} C_VEL
LIN {X 0,Y 214.147,Z 129.436,A -85,B 0,C 180,E1 -20690.55,E2 -20690.55} C_VEL
LIN {X 0,Y 214.091,Z 129.44,A -85,B 0,C 180,E1 -20694.342,E2 -20694.342} C_VEL
LIN {X 0,Y 214.421,Z 129.392,A -85,B 0,C 180,E1 -20698.116,E2 -20698.116} C_VEL
LIN {X 0,Y 214.549,Z 129.376,A -85,B 0,C 180,E1 -20699.994,E2 -20699.994} C_VEL
LIN {X 0,Y 214.449,Z 129.384,A -85,B 0,C 180,E1 -20701.872,E2 -20701.872} C_VEL
LIN {X 0,Y 214.18,Z 129.525,A -85,B 0,C 180,E1 -20706.825,E2 -20706.825} C_VEL
LIN {X 0,Y 215.06,Z 132.094,A -85,B 0,C 180,E1 -20707.977,E2 -20707.977} C_VEL
LIN {X 0,Y 217.263,Z 134.491,A -85,B 0,C 180,E1 -20710.086,E2 -20710.086} C_VEL
LIN {X 0,Y 219.165,Z 135.571,A -85,B 0,C 180,E1 -20711.614,E2 -20711.614} C_VEL
LIN {X 0,Y 220.623,Z 138.493,A -85,B 0,C 180,E1 -20712.878,E2 -20712.878} C_VEL
LIN {X 0,Y 223.393,Z 140.88,A -85,B 0,C 180,E1 -20714.803,E2 -20714.803} C_VEL
LIN {X 0,Y 224.098,Z 141.697,A -85,B 0,C 180,E1 -20715.279,E2 -20715.279} C_VEL
LIN {X 0,Y 226.223,Z 144.904,A -85,B 0,C 180,E1 -20716.694,E2 -20716.694} C_VEL
LIN {X 0,Y 228.256,Z 146.823,A -85,B 0,C 180,E1 -20717.868,E2 -20717.868} C_VEL
LIN {X 0,Y 230.731,Z 150.288,A -85,B 0,C 180,E1 -20719.284,E2 -20719.284} C_VEL
LIN {X 0,Y 232.404,Z 152.115,A -85,B 0,C 180,E1 -20720.156,E2 -20720.156} C_VEL
LIN {X 0,Y 235.386,Z 155.939,A -85,B 0,C 180,E1 -20721.66,E2 -20721.66} C_VEL
LIN {X 0,Y 240.676,Z 163.286,A -85,B 0,C 180,E1 -20724.123,E2 -20724.123} C_VEL
LIN {X 0,Y 244.803,Z 169.305,A -85,B 0,C 180,E1 -20725.871,E2 -20725.871} C_VEL
LIN {X 0,Y 251.197,Z 180.105,A -85,B 0,C 180,E1 -20728.393,E2 -20728.393} C_VEL
LIN {X 0,Y 257.391,Z 192.031,A -85,B 0,C 180,E1 -20730.645,E2 -20730.645} C_VEL
LIN {X 0,Y 260.168,Z 198.03,A -85,B 0,C 180,E1 -20731.614,E2 -20731.614} C_VEL
LIN {X 0,Y 256.096,Z 262.21,A -85,B 0,C 180,E1 -20733.346,E2 -20733.346} C_VEL
LIN {X 0,Y 254.279,Z 276.463,A -85,B 0,C 180,E1 -20733.983,E2 -20733.983} C_VEL
LIN {X 0,Y 251.959,Z 289.198,A -85,B 0,C 180,E1 -20734.8,E2 -20734.8} C_VEL
LIN {X 0,Y 248.971,Z 302.466,A -85,B 0,C 180,E1 -20735.981,E2 -20735.981} C_VEL
LIN {X 0,Y 245.523,Z 314.808,A -85,B 0,C 180,E1 -20737.405,E2 -20737.405} C_VEL
LIN {X 0,Y 241.362,Z 326.998,A -85,B 0,C 180,E1 -20739.167,E2 -20739.167} C_VEL
LIN {X 0,Y 237.445,Z 337.203,A -85,B 0,C 180,E1 -20741.04,E2 -20741.04} C_VEL
LIN {X 0,Y 233.476,Z 346.403,A -85,B 0,C 180,E1 -20743.113,E2 -20743.113} C_VEL
LIN {X 0,Y 229.089,Z 355.72,A -85,B 0,C 180,E1 -20745.736,E2 -20745.736} C_VEL
LIN {X 0,Y 225.079,Z 363.562,A -85,B 0,C 180,E1 -20748.526,E2 -20748.526} C_VEL
LIN {X 0,Y 221.247,Z 370.585,A -85,B 0,C 180,E1 -20751.723,E2 -20751.723} C_VEL
LIN {X 0,Y 218.4,Z 375.469,A -85,B 0,C 180,E1 -20754.601,E2 -20754.601} C_VEL
LIN {X 0,Y 215.96,Z 379.591,A -85,B 0,C 180,E1 -20757.778,E2 -20757.778} C_VEL
LIN {X 0,Y 214.296,Z 382.264,A -85,B 0,C 180,E1 -20760.529,E2 -20760.529} C_VEL
LIN {X 0,Y 212.559,Z 384.742,A -85,B 0,C 180,E1 -20764.541,E2 -20764.541} C_VEL
LIN {X 0,Y 211.58,Z 385.744,A -85,B 0,C 180,E1 -20768.566,E2 -20768.566} C_VEL
LIN {X 0,Y 211.128,Z 385.312,A -85,B 0,C 180,E1 -20772.564,E2 -20772.564} C_VEL
LIN {X 0,Y 211.125,Z 384.44,A -85,B 0,C 180,E1 -20774.844,E2 -20774.844} C_VEL
LIN {X 0,Y 211.267,Z 382.023,A -85,B 0,C 180,E1 -20778.484,E2 -20778.484} C_VEL
LIN {X 0,Y 211.755,Z 379.118,A -85,B 0,C 180,E1 -20781.408,E2 -20781.408} C_VEL
LIN {X 0,Y 212.423,Z 375.393,A -85,B 0,C 180,E1 -20784.301,E2 -20784.301} C_VEL
LIN {X 0,Y 213.289,Z 370.752,A -85,B 0,C 180,E1 -20787.164,E2 -20787.164} C_VEL
LIN {X 0,Y 214.825,Z 364.01,A -85,B 0,C 180,E1 -20790.466,E2 -20790.466} C_VEL
LIN {X 0,Y 216.925,Z 355.607,A -85,B 0,C 180,E1 -20793.713,E2 -20793.713} C_VEL
LIN {X 0,Y 219.315,Z 346.076,A -85,B 0,C 180,E1 -20796.656,E2 -20796.656} C_VEL
LIN {X 0,Y 221.609,Z 336.273,A -85,B 0,C 180,E1 -20799.121,E2 -20799.121} C_VEL
LIN {X 0,Y 223.837,Z 326.752,A -85,B 0,C 180,E1 -20801.085,E2 -20801.085} C_VEL
LIN {X 0,Y 226.278,Z 315.327,A -85,B 0,C 180,E1 -20803.011,E2 -20803.011} C_VEL
LIN {X 0,Y 228.627,Z 302.826,A -85,B 0,C 180,E1 -20804.688,E2 -20804.688} C_VEL
LIN {X 0,Y 230.643,Z 289.991,A -85,B 0,C 180,E1 -20806.028,E2 -20806.028} C_VEL
LIN {X 0,Y 232.329,Z 275.589,A -85,B 0,C 180,E1 -20807.151,E2 -20807.151} C_VEL
LIN {X 0,Y 233.5,Z 261.227,A -85,B 0,C 180,E1 -20807.91,E2 -20807.91} C_VEL
LIN {X 0,Y 237.354,Z 178.541,A -85,B 0,C 180,E1 -20810.326,E2 -20810.326} C_VEL
LIN {X 0,Y 230.442,Z 160.544,A -85,B 0,C 180,E1 -20812.011,E2 -20812.011} C_VEL
LIN {X 0,Y 224.975,Z 149.489,A -85,B 0,C 180,E1 -20813.317,E2 -20813.317} C_VEL
LIN {X 0,Y 217.492,Z 136.52,A -85,B 0,C 180,E1 -20815.148,E2 -20815.148} C_VEL
LIN {X 0,Y 215.509,Z 133.265,A -85,B 0,C 180,E1 -20815.654,E2 -20815.654} C_VEL
LIN {X 0,Y 214.02,Z 130.507,A -85,B 0,C 180,E1 -20816.055,E2 -20816.055} C_VEL
LIN {X 0,Y 213.818,Z 129.472,A -85,B 0,C 180,E1 -20816.192,E2 -20816.192} C_VEL
LIN {X 0,Y 213.766,Z 129.482,A -85,B 0,C 180,E1 -20821.277,E2 -20821.277} C_VEL
LIN {X 0,Y 213.758,Z 129.482,A -85,B 0,C 180,E1 -20826.282,E2 -20826.282} C_VEL
LIN {X 0,Y 213.807,Z 129.474,A -85,B 0,C 180,E1 -20831.099,E2 -20831.099} C_VEL
LIN {X 0,Y 213.809,Z 129.455,A -85,B 0,C 180,E1 -20833.696,E2 -20833.696} C_VEL
LIN {X 0,Y 213.814,Z 129.471,A -85,B 0,C 180,E1 -20836.359,E2 -20836.359} C_VEL
LIN {X 0,Y 213.798,Z 129.47,A -85,B 0,C 180,E1 -20839.114,E2 -20839.114} C_VEL
LIN {X 0,Y 213.73,Z 129.473,A -85,B 0,C 180,E1 -20843.718,E2 -20843.718} C_VEL
LIN {X 0,Y 213.747,Z 129.476,A -85,B 0,C 180,E1 -20848.268,E2 -20848.268} C_VEL
LIN {X 0,Y 213.805,Z 129.45,A -85,B 0,C 180,E1 -20852.608,E2 -20852.608} C_VEL
LIN {X 0,Y 213.851,Z 129.471,A -85,B 0,C 180,E1 -20856.947,E2 -20856.947} C_VEL
LIN {X 0,Y 213.923,Z 129.463,A -85,B 0,C 180,E1 -20862.304,E2 -20862.304} C_VEL
LIN {X 0,Y 213.966,Z 129.453,A -85,B 0,C 180,E1 -20866.714,E2 -20866.714} C_VEL
LIN {X 0,Y 214.182,Z 129.421,A -85,B 0,C 180,E1 -20870.564,E2 -20870.564} C_VEL
LIN {X 0,Y 214.1,Z 129.409,A -85,B 0,C 180,E1 -20874.355,E2 -20874.355} C_VEL
LIN {X 0,Y 214.438,Z 129.396,A -85,B 0,C 180,E1 -20878.128,E2 -20878.128} C_VEL
LIN {X 0,Y 214.545,Z 129.382,A -85,B 0,C 180,E1 -20880.006,E2 -20880.006} C_VEL
LIN {X 0,Y 214.437,Z 129.387,A -85,B 0,C 180,E1 -20881.884,E2 -20881.884} C_VEL
LIN {X 0,Y 214.221,Z 129.417,A -85,B 0,C 180,E1 -20887.547,E2 -20887.547} C_VEL
LIN {X 0,Y 214.039,Z 129.444,A -85,B 0,C 180,E1 -20891.368,E2 -20891.368} C_VEL
LIN {X 0,Y 213.929,Z 129.461,A -85,B 0,C 180,E1 -20895.243,E2 -20895.243} C_VEL
LIN {X 0,Y 213.837,Z 129.474,A -85,B 0,C 180,E1 -20899.193,E2 -20899.193} C_VEL
LIN {X 0,Y 213.846,Z 129.47,A -85,B 0,C 180,E1 -20903.233,E2 -20903.233} C_VEL
LIN {X 0,Y 213.802,Z 129.466,A -85,B 0,C 180,E1 -20907.787,E2 -20907.787} C_VEL
LIN {X 0,Y 213.769,Z 129.475,A -85,B 0,C 180,E1 -20911.743,E2 -20911.743} C_VEL
LIN {X 0,Y 213.739,Z 129.484,A -85,B 0,C 180,E1 -20915.957,E2 -20915.957} C_VEL
LIN {X 0,Y 213.426,Z 129.527,A -85,B 0,C 180,E1 -20917.009,E2 -20917.009} C_VEL
LIN {X 0,Y 212.058,Z 129.699,A -85,B 0,C 180,E1 -20918.562,E2 -20918.562} C_VEL
LIN {X 0,Y 207.698,Z 130.235,A -85,B 0,C 180,E1 -20922.194,E2 -20922.194} C_VEL
LIN {X 0,Y 206.71,Z 130.361,A -85,B 0,C 180,E1 -20923.827,E2 -20923.827} C_VEL
LIN {X 0,Y 206.663,Z 130.367,A -85,B 0,C 180,E1 -20924.38,E2 -20924.38} C_VEL
LIN {X 0,Y 206.729,Z 130.505,A -85,B 0,C 180,E1 -20924.906,E2 -20924.906} C_VEL
LIN {X 0,Y 207.533,Z 133.624,A -85,B 0,C 180,E1 -20926.397,E2 -20926.397} C_VEL
LIN {X 0,Y 216.137,Z 150.248,A -85,B 0,C 180,E1 -20928.782,E2 -20928.782} C_VEL
LIN {X 0,Y 223.293,Z 166.773,A -85,B 0,C 180,E1 -20930.697,E2 -20930.697} C_VEL
LIN {X 0,Y 229.107,Z 182.247,A -85,B 0,C 180,E1 -20932.213,E2 -20932.213} C_VEL
LIN {X 0,Y 230.696,Z 194.994,A -85,B 0,C 180,E1 -20932.919,E2 -20932.919} C_VEL
LIN {X 0,Y 227.188,Z 271.667,A -85,B 0,C 180,E1 -20935.228,E2 -20935.228} C_VEL
LIN {X 0,Y 225.795,Z 286.481,A -85,B 0,C 180,E1 -20935.997,E2 -20935.997} C_VEL
LIN {X 0,Y 224.023,Z 299.431,A -85,B 0,C 180,E1 -20936.973,E2 -20936.973} C_VEL
LIN {X 0,Y 221.941,Z 311.896,A -85,B 0,C 180,E1 -20938.237,E2 -20938.237} C_VEL
LIN {X 0,Y 219.516,Z 324.292,A -85,B 0,C 180,E1 -20939.866,E2 -20939.866} C_VEL
LIN {X 0,Y 216.919,Z 335.589,A -85,B 0,C 180,E1 -20941.719,E2 -20941.719} C_VEL
LIN {X 0,Y 214.623,Z 345.646,A -85,B 0,C 180,E1 -20943.767,E2 -20943.767} C_VEL
LIN {X 0,Y 212.124,Z 355.011,A -85,B 0,C 180,E1 -20946.058,E2 -20946.058} C_VEL
LIN {X 0,Y 209.752,Z 364.39,A -85,B 0,C 180,E1 -20948.891,E2 -20948.891} C_VEL
LIN {X 0,Y 207.859,Z 372.112,A -85,B 0,C 180,E1 -20951.746,E2 -20951.746} C_VEL
LIN {X 0,Y 206.245,Z 379.596,A -85,B 0,C 180,E1 -20955.196,E2 -20955.196} C_VEL
LIN {X 0,Y 205.207,Z 384.764,A -85,B 0,C 180,E1 -20958.145,E2 -20958.145} C_VEL
LIN {X 0,Y 204.651,Z 388.889,A -85,B 0,C 180,E1 -20961.113,E2 -20961.113} C_VEL
LIN {X 0,Y 204.399,Z 392.134,A -85,B 0,C 180,E1 -20964.082,E2 -20964.082} C_VEL
LIN {X 0,Y 204.373,Z 395.14,A -85,B 0,C 180,E1 -20968.032,E2 -20968.032} C_VEL
LIN {X 0,Y 204.488,Z 396.114,A -85,B 0,C 180,E1 -20970.003,E2 -20970.003} C_VEL
LIN {X 0,Y 204.337,Z 397.031,A -85,B 0,C 180,E1 -20974.047,E2 -20974.047} C_VEL
LIN {X 0,Y 204.574,Z 396.614,A -85,B 0,C 180,E1 -20977.901,E2 -20977.901} C_VEL
LIN {X 0,Y 205.444,Z 394.902,A -85,B 0,C 180,E1 -20981.847,E2 -20981.847} C_VEL
LIN {X 0,Y 207.15,Z 391.857,A -85,B 0,C 180,E1 -20985.751,E2 -20985.751} C_VEL
LIN {X 0,Y 209.755,Z 387.4,A -85,B 0,C 180,E1 -20989.579,E2 -20989.579} C_VEL
LIN {X 0,Y 213.083,Z 381.399,A -85,B 0,C 180,E1 -20993.318,E2 -20993.318} C_VEL
LIN {X 0,Y 216.866,Z 374.693,A -85,B 0,C 180,E1 -20996.464,E2 -20996.464} C_VEL
LIN {X 0,Y 221.326,Z 366.391,A -85,B 0,C 180,E1 -20999.487,E2 -20999.487} C_VEL
LIN {X 0,Y 225.726,Z 357.772,A -85,B 0,C 180,E1 -21001.961,E2 -21001.961} C_VEL
LIN {X 0,Y 230.179,Z 347.719,A -85,B 0,C 180,E1 -21004.308,E2 -21004.308} C_VEL
LIN {X 0,Y 234.681,Z 336.968,A -85,B 0,C 180,E1 -21006.263,E2 -21006.263} C_VEL
LIN {X 0,Y 238.779,Z 325.661,A -85,B 0,C 180,E1 -21007.912,E2 -21007.912} C_VEL
LIN {X 0,Y 242.551,Z 313.334,A -85,B 0,C 180,E1 -21009.336,E2 -21009.336} C_VEL
LIN {X 0,Y 246.12,Z 299.571,A -85,B 0,C 180,E1 -21010.516,E2 -21010.516} C_VEL
LIN {X 0,Y 248.858,Z 285.783,A -85,B 0,C 180,E1 -21011.38,E2 -21011.38} C_VEL
LIN {X 0,Y 250.778,Z 271.543,A -85,B 0,C 180,E1 -21012,E2 -21012} C_VEL
LIN {X 0,Y 255.026,Z 208.096,A -85,B 0,C 180,E1 -21013.703,E2 -21013.703} C_VEL
LIN {X 0,Y 252.416,Z 201.658,A -85,B 0,C 180,E1 -21014.694,E2 -21014.694} C_VEL
LIN {X 0,Y 246.83,Z 189.716,A -85,B 0,C 180,E1 -21016.888,E2 -21016.888} C_VEL
LIN {X 0,Y 240.266,Z 177.57,A -85,B 0,C 180,E1 -21019.67,E2 -21019.67} C_VEL
LIN {X 0,Y 234.011,Z 167.146,A -85,B 0,C 180,E1 -21022.656,E2 -21022.656} C_VEL
LIN {X 0,Y 230.046,Z 161.16,A -85,B 0,C 180,E1 -21024.743,E2 -21024.743} C_VEL
LIN {X 0,Y 226.886,Z 156.396,A -85,B 0,C 180,E1 -21026.569,E2 -21026.569} C_VEL
LIN {X 0,Y 222.503,Z 150.254,A -85,B 0,C 180,E1 -21029.386,E2 -21029.386} C_VEL
LIN {X 0,Y 219.18,Z 145.968,A -85,B 0,C 180,E1 -21031.833,E2 -21031.833} C_VEL
LIN {X 0,Y 218.121,Z 144.32,A -85,B 0,C 180,E1 -21032.722,E2 -21032.722} C_VEL
LIN {X 0,Y 214.769,Z 140.646,A -85,B 0,C 180,E1 -21035.72,E2 -21035.72} C_VEL
LIN {X 0,Y 213.017,Z 138.266,A -85,B 0,C 180,E1 -21037.621,E2 -21037.621} C_VEL
LIN {X 0,Y 212.373,Z 137.054,A -85,B 0,C 180,E1 -21038.444,E2 -21038.444} C_VEL
LIN {X 0,Y 211.472,Z 136.147,A -85,B 0,C 180,E1 -21039.571,E2 -21039.571} C_VEL
LIN {X 0,Y 208.245,Z 133.69,A -85,B 0,C 180,E1 -21044.832,E2 -21044.832} C_VEL
LIN {X 0,Y 207.081,Z 130.684,A -85,B 0,C 180,E1 -21049.454,E2 -21049.454} C_VEL
LIN {X 0,Y 207.102,Z 130.313,A -85,B 0,C 180,E1 -21050.225,E2 -21050.225} C_VEL
LIN {X 0,Y 207.066,Z 130.337,A -85,B 0,C 180,E1 -21054.638,E2 -21054.638} C_VEL
LIN {X 0,Y 207.634,Z 131.835,A -85,B 0,C 180,E1 -21057.569,E2 -21057.569} C_VEL
LIN {X 0,Y 209.596,Z 134.619,A -85,B 0,C 180,E1 -21062.155,E2 -21062.155} C_VEL
LIN {X 0,Y 211.683,Z 136.111,A -85,B 0,C 180,E1 -21065.088,E2 -21065.088} C_VEL
LIN {X 0,Y 212.727,Z 136.527,A -85,B 0,C 180,E1 -21066.276,E2 -21066.276} C_VEL
LIN {X 0,Y 213.919,Z 139.247,A -85,B 0,C 180,E1 -21067.782,E2 -21067.782} C_VEL
LIN {X 0,Y 216.358,Z 141.637,A -85,B 0,C 180,E1 -21070.111,E2 -21070.111} C_VEL
LIN {X 0,Y 217.505,Z 142.422,A -85,B 0,C 180,E1 -21071.065,E2 -21071.065} C_VEL
LIN {X 0,Y 219.137,Z 145.33,A -85,B 0,C 180,E1 -21072.496,E2 -21072.496} C_VEL
LIN {X 0,Y 222.075,Z 148.015,A -85,B 0,C 180,E1 -21074.6,E2 -21074.6} C_VEL
LIN {X 0,Y 224.337,Z 151.425,A -85,B 0,C 180,E1 -21076.165,E2 -21076.165} C_VEL
LIN {X 0,Y 226.254,Z 153.437,A -85,B 0,C 180,E1 -21077.323,E2 -21077.323} C_VEL
LIN {X 0,Y 229.17,Z 157.244,A -85,B 0,C 180,E1 -21079.014,E2 -21079.014} C_VEL
LIN {X 0,Y 230.352,Z 158.777,A -85,B 0,C 180,E1 -21079.661,E2 -21079.661} C_VEL
LIN {X 0,Y 234.029,Z 163.682,A -85,B 0,C 180,E1 -21081.563,E2 -21081.563} C_VEL
LIN {X 0,Y 239.217,Z 170.929,A -85,B 0,C 180,E1 -21084.008,E2 -21084.008} C_VEL
LIN {X 0,Y 242.507,Z 176.249,A -85,B 0,C 180,E1 -21085.458,E2 -21085.458} C_VEL
LIN {X 0,Y 248.006,Z 185.764,A -85,B 0,C 180,E1 -21087.704,E2 -21087.704} C_VEL
LIN {X 0,Y 253.754,Z 197.17,A -85,B 0,C 180,E1 -21089.896,E2 -21089.896} C_VEL
LIN {X 0,Y 255.352,Z 200.736,A -85,B 0,C 180,E1 -21090.484,E2 -21090.484} C_VEL
LIN {X 0,Y 251.342,Z 261.882,A -85,B 0,C 180,E1 -21092.144,E2 -21092.144} C_VEL
LIN {X 0,Y 249.503,Z 276.26,A -85,B 0,C 180,E1 -21092.789,E2 -21092.789} C_VEL
LIN {X 0,Y 246.953,Z 289.677,A -85,B 0,C 180,E1 -21093.648,E2 -21093.648} C_VEL
LIN {X 0,Y 243.948,Z 302.561,A -85,B 0,C 180,E1 -21094.806,E2 -21094.806} C_VEL
LIN {X 0,Y 240.516,Z 314.424,A -85,B 0,C 180,E1 -21096.172,E2 -21096.172} C_VEL
LIN {X 0,Y 236.207,Z 326.711,A -85,B 0,C 180,E1 -21097.954,E2 -21097.954} C_VEL
LIN {X 0,Y 232.208,Z 336.703,A -85,B 0,C 180,E1 -21099.78,E2 -21099.78} C_VEL
LIN {X 0,Y 227.559,Z 347.103,A -85,B 0,C 180,E1 -21102.161,E2 -21102.161} C_VEL
LIN {X 0,Y 222.985,Z 356.328,A -85,B 0,C 180,E1 -21104.831,E2 -21104.831} C_VEL
LIN {X 0,Y 218.9,Z 363.903,A -85,B 0,C 180,E1 -21107.603,E2 -21107.603} C_VEL
LIN {X 0,Y 215.311,Z 370.104,A -85,B 0,C 180,E1 -21110.465,E2 -21110.465} C_VEL
LIN {X 0,Y 212.238,Z 375.136,A -85,B 0,C 180,E1 -21113.41,E2 -21113.41} C_VEL
LIN {X 0,Y 209.263,Z 379.848,A -85,B 0,C 180,E1 -21117.084,E2 -21117.084} C_VEL
LIN {X 0,Y 207.706,Z 382.167,A -85,B 0,C 180,E1 -21119.497,E2 -21119.497} C_VEL
LIN {X 0,Y 205.78,Z 384.797,A -85,B 0,C 180,E1 -21123.638,E2 -21123.638} C_VEL
LIN {X 0,Y 204.625,Z 385.918,A -85,B 0,C 180,E1 -21127.799,E2 -21127.799} C_VEL
LIN {X 0,Y 204.063,Z 385.605,A -85,B 0,C 180,E1 -21131.94,E2 -21131.94} C_VEL
LIN {X 0,Y 204.024,Z 384.644,A -85,B 0,C 180,E1 -21134.659,E2 -21134.659} C_VEL
LIN {X 0,Y 204.129,Z 382.491,A -85,B 0,C 180,E1 -21138.076,E2 -21138.076} C_VEL
LIN {X 0,Y 204.807,Z 378.616,A -85,B 0,C 180,E1 -21142.108,E2 -21142.108} C_VEL
LIN {X 0,Y 205.528,Z 374.664,A -85,B 0,C 180,E1 -21145.093,E2 -21145.093} C_VEL
LIN {X 0,Y 206.536,Z 369.797,A -85,B 0,C 180,E1 -21148.047,E2 -21148.047} C_VEL
LIN {X 0,Y 208.241,Z 362.764,A -85,B 0,C 180,E1 -21151.448,E2 -21151.448} C_VEL
LIN {X 0,Y 210.493,Z 354.054,A -85,B 0,C 180,E1 -21154.785,E2 -21154.785} C_VEL
LIN {X 0,Y 212.868,Z 344.949,A -85,B 0,C 180,E1 -21157.586,E2 -21157.586} C_VEL
LIN {X 0,Y 215.041,Z 335.913,A -85,B 0,C 180,E1 -21159.877,E2 -21159.877} C_VEL
LIN {X 0,Y 217.69,Z 325.086,A -85,B 0,C 180,E1 -21162.111,E2 -21162.111} C_VEL
LIN {X 0,Y 220.23,Z 313.27,A -85,B 0,C 180,E1 -21164.08,E2 -21164.08} C_VEL
LIN {X 0,Y 222.683,Z 300.238,A -85,B 0,C 180,E1 -21165.793,E2 -21165.793} C_VEL
LIN {X 0,Y 224.804,Z 286.571,A -85,B 0,C 180,E1 -21167.157,E2 -21167.157} C_VEL
LIN {X 0,Y 226.381,Z 272.219,A -85,B 0,C 180,E1 -21168.201,E2 -21168.201} C_VEL
LIN {X 0,Y 227.478,Z 258.148,A -85,B 0,C 180,E1 -21168.868,E2 -21168.868} C_VEL
LIN {X 0,Y 231.252,Z 180.926,A -85,B 0,C 180,E1 -21171.141,E2 -21171.141} C_VEL
LIN {X 0,Y 228.813,Z 173.796,A -85,B 0,C 180,E1 -21171.778,E2 -21171.778} C_VEL
LIN {X 0,Y 223.655,Z 160.913,A -85,B 0,C 180,E1 -21173.102,E2 -21173.102} C_VEL
LIN {X 0,Y 216.649,Z 147.783,A -85,B 0,C 180,E1 -21174.849,E2 -21174.849} C_VEL
LIN {X 0,Y 210.502,Z 137.476,A -85,B 0,C 180,E1 -21176.461,E2 -21176.461} C_VEL
LIN {X 0,Y 208.609,Z 134.287,A -85,B 0,C 180,E1 -21176.984,E2 -21176.984} C_VEL
LIN {X 0,Y 207.056,Z 131.686,A -85,B 0,C 180,E1 -21177.422,E2 -21177.422} C_VEL
LIN {X 0,Y 206.758,Z 130.346,A -85,B 0,C 180,E1 -21177.606,E2 -21177.606} C_VEL
LIN {X 0,Y 206.699,Z 130.363,A -85,B 0,C 180,E1 -21181.801,E2 -21181.801} C_VEL
LIN {X 0,Y 206.721,Z 130.358,A -85,B 0,C 180,E1 -21185.333,E2 -21185.333} C_VEL
LIN {X 0,Y 206.729,Z 130.359,A -85,B 0,C 180,E1 -21190.231,E2 -21190.231} C_VEL
LIN {X 0,Y 206.718,Z 130.339,A -85,B 0,C 180,E1 -21194.453,E2 -21194.453} C_VEL
LIN {X 0,Y 206.724,Z 130.356,A -85,B 0,C 180,E1 -21198.407,E2 -21198.407} C_VEL
LIN {X 0,Y 206.7,Z 130.334,A -85,B 0,C 180,E1 -21202.274,E2 -21202.274} C_VEL
LIN {X 0,Y 206.682,Z 130.361,A -85,B 0,C 180,E1 -21207.048,E2 -21207.048} C_VEL
LIN {X 0,Y 206.743,Z 130.324,A -85,B 0,C 180,E1 -21212.103,E2 -21212.103} C_VEL
LIN {X 0,Y 206.78,Z 130.353,A -85,B 0,C 180,E1 -21216.58,E2 -21216.58} C_VEL
LIN {X 0,Y 206.869,Z 130.342,A -85,B 0,C 180,E1 -21222.026,E2 -21222.026} C_VEL
LIN {X 0,Y 206.899,Z 130.332,A -85,B 0,C 180,E1 -21226.252,E2 -21226.252} C_VEL
LIN {X 0,Y 207.118,Z 130.302,A -85,B 0,C 180,E1 -21230.239,E2 -21230.239} C_VEL
LIN {X 0,Y 207.063,Z 130.283,A -85,B 0,C 180,E1 -21234.162,E2 -21234.162} C_VEL
LIN {X 0,Y 207.375,Z 130.276,A -85,B 0,C 180,E1 -21238.064,E2 -21238.064} C_VEL
LIN {X 0,Y 207.509,Z 130.258,A -85,B 0,C 180,E1 -21240.006,E2 -21240.006} C_VEL
LIN {X 0,Y 207.076,Z 130.285,A -85,B 0,C 180,E1 -21243.898,E2 -21243.898} C_VEL
LIN {X 0,Y 207.161,Z 130.298,A -85,B 0,C 180,E1 -21247.805,E2 -21247.805} C_VEL
LIN {X 0,Y 206.976,Z 130.322,A -85,B 0,C 180,E1 -21251.761,E2 -21251.761} C_VEL
LIN {X 0,Y 206.863,Z 130.34,A -85,B 0,C 180,E1 -21255.777,E2 -21255.777} C_VEL
LIN {X 0,Y 206.781,Z 130.352,A -85,B 0,C 180,E1 -21259.875,E2 -21259.875} C_VEL
LIN {X 0,Y 206.762,Z 130.352,A -85,B 0,C 180,E1 -21264.078,E2 -21264.078} C_VEL
LIN {X 0,Y 206.744,Z 130.347,A -85,B 0,C 180,E1 -21268.425,E2 -21268.425} C_VEL
LIN {X 0,Y 206.7,Z 130.355,A -85,B 0,C 180,E1 -21272.964,E2 -21272.964} C_VEL
LIN {X 0,Y 206.678,Z 130.365,A -85,B 0,C 180,E1 -21277.747,E2 -21277.747} C_VEL
LIN {X 0,Y 206.64,Z 130.36,A -85,B 0,C 180,E1 -21281.567,E2 -21281.567} C_VEL
LIN {X 0,Y 206.663,Z 130.367,A -85,B 0,C 180,E1 -21284.38,E2 -21284.38} C_VEL
LIN {X 0,Y 206.902,Z 131.228,A -85,B 0,C 180,E1 -21285.195,E2 -21285.195} C_VEL
LIN {X 0,Y 207.507,Z 133.918,A -85,B 0,C 180,E1 -21286.023,E2 -21286.023} C_VEL
LIN {X 0,Y 208.491,Z 138.993,A -85,B 0,C 180,E1 -21286.79,E2 -21286.79} C_VEL
LIN {X 0,Y 210.144,Z 149.551,A -85,B 0,C 180,E1 -21287.607,E2 -21287.607} C_VEL
LIN {X 0,Y 211.763,Z 155.757,A -85,B 0,C 180,E1 -21288.181,E2 -21288.181} C_VEL
LIN {X 0,Y 212.609,Z 157.638,A -85,B 0,C 180,E1 -21288.422,E2 -21288.422} C_VEL
LIN {X 0,Y 219.81,Z 175.244,A -85,B 0,C 180,E1 -21290.433,E2 -21290.433} C_VEL
LIN {X 0,Y 223.498,Z 185.357,A -85,B 0,C 180,E1 -21291.44,E2 -21291.44} C_VEL
LIN {X 0,Y 224.597,Z 196.315,A -85,B 0,C 180,E1 -21292.031,E2 -21292.031} C_VEL
LIN {X 0,Y 220.946,Z 272.261,A -85,B 0,C 180,E1 -21294.377,E2 -21294.377} C_VEL
LIN {X 0,Y 219.492,Z 286.793,A -85,B 0,C 180,E1 -21295.159,E2 -21295.159} C_VEL
LIN {X 0,Y 217.672,Z 299.615,A -85,B 0,C 180,E1 -21296.158,E2 -21296.158} C_VEL
LIN {X 0,Y 215.524,Z 311.999,A -85,B 0,C 180,E1 -21297.453,E2 -21297.453} C_VEL
LIN {X 0,Y 212.997,Z 324.397,A -85,B 0,C 180,E1 -21299.129,E2 -21299.129} C_VEL
LIN {X 0,Y 210.329,Z 335.593,A -85,B 0,C 180,E1 -21301.023,E2 -21301.023} C_VEL
LIN {X 0,Y 207.641,Z 346.602,A -85,B 0,C 180,E1 -21303.358,E2 -21303.358} C_VEL
LIN {X 0,Y 205.121,Z 355.783,A -85,B 0,C 180,E1 -21305.726,E2 -21305.726} C_VEL
LIN {X 0,Y 202.678,Z 364.999,A -85,B 0,C 180,E1 -21308.651,E2 -21308.651} C_VEL
LIN {X 0,Y 200.765,Z 372.656,A -85,B 0,C 180,E1 -21311.639,E2 -21311.639} C_VEL
LIN {X 0,Y 199.313,Z 379.021,A -85,B 0,C 180,E1 -21314.668,E2 -21314.668} C_VEL
LIN {X 0,Y 198.191,Z 384.236,A -85,B 0,C 180,E1 -21317.719,E2 -21317.719} C_VEL
LIN {X 0,Y 197.608,Z 388.438,A -85,B 0,C 180,E1 -21320.794,E2 -21320.794} C_VEL
LIN {X 0,Y 197.315,Z 391.755,A -85,B 0,C 180,E1 -21323.869,E2 -21323.869} C_VEL
LIN {X 0,Y 197.279,Z 394.829,A -85,B 0,C 180,E1 -21327.961,E2 -21327.961} C_VEL
LIN {X 0,Y 197.407,Z 395.836,A -85,B 0,C 180,E1 -21330.003,E2 -21330.003} C_VEL
LIN {X 0,Y 197.262,Z 396.811,A -85,B 0,C 180,E1 -21334.089,E2 -21334.089} C_VEL
LIN {X 0,Y 197.512,Z 396.467,A -85,B 0,C 180,E1 -21338.186,E2 -21338.186} C_VEL
LIN {X 0,Y 198.47,Z 394.821,A -85,B 0,C 180,E1 -21342.27,E2 -21342.27} C_VEL
LIN {X 0,Y 200.29,Z 391.846,A -85,B 0,C 180,E1 -21346.306,E2 -21346.306} C_VEL
LIN {X 0,Y 203.053,Z 387.461,A -85,B 0,C 180,E1 -21350.253,E2 -21350.253} C_VEL
LIN {X 0,Y 206.565,Z 381.551,A -85,B 0,C 180,E1 -21354.1,E2 -21354.1} C_VEL
LIN {X 0,Y 210.529,Z 374.942,A -85,B 0,C 180,E1 -21357.326,E2 -21357.326} C_VEL
LIN {X 0,Y 215.182,Z 366.772,A -85,B 0,C 180,E1 -21360.417,E2 -21360.417} C_VEL
LIN {X 0,Y 219.758,Z 358.275,A -85,B 0,C 180,E1 -21362.937,E2 -21362.937} C_VEL
LIN {X 0,Y 224.628,Z 347.826,A -85,B 0,C 180,E1 -21365.431,E2 -21365.431} C_VEL
LIN {X 0,Y 229.026,Z 337.781,A -85,B 0,C 180,E1 -21367.308,E2 -21367.308} C_VEL
LIN {X 0,Y 233.277,Z 326.685,A -85,B 0,C 180,E1 -21368.972,E2 -21368.972} C_VEL
LIN {X 0,Y 237.16,Z 314.648,A -85,B 0,C 180,E1 -21370.412,E2 -21370.412} C_VEL
LIN {X 0,Y 240.86,Z 301.292,A -85,B 0,C 180,E1 -21371.594,E2 -21371.594} C_VEL
LIN {X 0,Y 243.77,Z 287.432,A -85,B 0,C 180,E1 -21372.512,E2 -21372.512} C_VEL
LIN {X 0,Y 245.923,Z 272.95,A -85,B 0,C 180,E1 -21373.167,E2 -21373.167} C_VEL
LIN {X 0,Y 247.609,Z 250.61,A -85,B 0,C 180,E1 -21373.82,E2 -21373.82} C_VEL
LIN {X 0,Y 250.292,Z 210.339,A -85,B 0,C 180,E1 -21374.895,E2 -21374.895} C_VEL
LIN {X 0,Y 245.949,Z 200.294,A -85,B 0,C 180,E1 -21376.648,E2 -21376.648} C_VEL
LIN {X 0,Y 241.382,Z 190.854,A -85,B 0,C 180,E1 -21378.588,E2 -21378.588} C_VEL
LIN {X 0,Y 236.19,Z 181.329,A -85,B 0,C 180,E1 -21380.966,E2 -21380.966} C_VEL
LIN {X 0,Y 230.947,Z 172.377,A -85,B 0,C 180,E1 -21383.63,E2 -21383.63} C_VEL
LIN {X 0,Y 227.614,Z 167.158,A -85,B 0,C 180,E1 -21385.48,E2 -21385.48} C_VEL
LIN {X 0,Y 224.315,Z 162.121,A -85,B 0,C 180,E1 -21387.478,E2 -21387.478} C_VEL
LIN {X 0,Y 220.477,Z 156.572,A -85,B 0,C 180,E1 -21390.081,E2 -21390.081} C_VEL
LIN {X 0,Y 217.325,Z 152.297,A -85,B 0,C 180,E1 -21392.536,E2 -21392.536} C_VEL
LIN {X 0,Y 216.341,Z 150.781,A -85,B 0,C 180,E1 -21393.398,E2 -21393.398} C_VEL
LIN {X 0,Y 213.409,Z 147.453,A -85,B 0,C 180,E1 -21396.137,E2 -21396.137} C_VEL
LIN {X 0,Y 211.521,Z 144.769,A -85,B 0,C 180,E1 -21398.286,E2 -21398.286} C_VEL
LIN {X 0,Y 210.817,Z 143.56,A -85,B 0,C 180,E1 -21399.224,E2 -21399.224} C_VEL
LIN {X 0,Y 209.534,Z 142.748,A -85,B 0,C 180,E1 -21400.906,E2 -21400.906} C_VEL
LIN {X 0,Y 206.438,Z 139.144,A -85,B 0,C 180,E1 -21407.709,E2 -21407.709} C_VEL
LIN {X 0,Y 206.131,Z 137.327,A -85,B 0,C 180,E1 -21410.178,E2 -21410.178} C_VEL
LIN {X 0,Y 206.16,Z 137.535,A -85,B 0,C 180,E1 -21414.615,E2 -21414.615} C_VEL
LIN {X 0,Y 207.519,Z 140.12,A -85,B 0,C 180,E1 -21419.751,E2 -21419.751} C_VEL
LIN {X 0,Y 209.789,Z 142.687,A -85,B 0,C 180,E1 -21423.835,E2 -21423.835} C_VEL
LIN {X 0,Y 211.387,Z 143.52,A -85,B 0,C 180,E1 -21425.821,E2 -21425.821} C_VEL
LIN {X 0,Y 212.787,Z 146.353,A -85,B 0,C 180,E1 -21427.585,E2 -21427.585} C_VEL
LIN {X 0,Y 215.476,Z 148.772,A -85,B 0,C 180,E1 -21430.153,E2 -21430.153} C_VEL
LIN {X 0,Y 215.978,Z 149.362,A -85,B 0,C 180,E1 -21430.603,E2 -21430.603} C_VEL
LIN {X 0,Y 217.943,Z 152.48,A -85,B 0,C 180,E1 -21432.329,E2 -21432.329} C_VEL
LIN {X 0,Y 220.226,Z 154.61,A -85,B 0,C 180,E1 -21434.018,E2 -21434.018} C_VEL
LIN {X 0,Y 222.698,Z 158.183,A -85,B 0,C 180,E1 -21435.773,E2 -21435.773} C_VEL
LIN {X 0,Y 224.259,Z 159.978,A -85,B 0,C 180,E1 -21436.756,E2 -21436.756} C_VEL
LIN {X 0,Y 228.195,Z 165.192,A -85,B 0,C 180,E1 -21439.084,E2 -21439.084} C_VEL
LIN {X 0,Y 231.454,Z 169.616,A -85,B 0,C 180,E1 -21440.838,E2 -21440.838} C_VEL
LIN {X 0,Y 236.669,Z 177.105,A -85,B 0,C 180,E1 -21443.397,E2 -21443.397} C_VEL
LIN {X 0,Y 241.16,Z 184.685,A -85,B 0,C 180,E1 -21445.438,E2 -21445.438} C_VEL
LIN {X 0,Y 246.198,Z 194.015,A -85,B 0,C 180,E1 -21447.545,E2 -21447.545} C_VEL
LIN {X 0,Y 250.649,Z 203.418,A -85,B 0,C 180,E1 -21449.312,E2 -21449.312} C_VEL
LIN {X 0,Y 246.589,Z 262.727,A -85,B 0,C 180,E1 -21450.946,E2 -21450.946} C_VEL
LIN {X 0,Y 244.697,Z 276.855,A -85,B 0,C 180,E1 -21451.592,E2 -21451.592} C_VEL
LIN {X 0,Y 242.051,Z 290.156,A -85,B 0,C 180,E1 -21452.449,E2 -21452.449} C_VEL
LIN {X 0,Y 238.696,Z 303.912,A -85,B 0,C 180,E1 -21453.715,E2 -21453.715} C_VEL
LIN {X 0,Y 235.058,Z 315.804,A -85,B 0,C 180,E1 -21455.125,E2 -21455.125} C_VEL
LIN {X 0,Y 230.689,Z 327.675,A -85,B 0,C 180,E1 -21456.894,E2 -21456.894} C_VEL
LIN {X 0,Y 226.039,Z 338.692,A -85,B 0,C 180,E1 -21458.982,E2 -21458.982} C_VEL
LIN {X 0,Y 221.756,Z 347.709,A -85,B 0,C 180,E1 -21461.125,E2 -21461.125} C_VEL
LIN {X 0,Y 216.945,Z 356.959,A -85,B 0,C 180,E1 -21463.877,E2 -21463.877} C_VEL
LIN {X 0,Y 212.842,Z 364.139,A -85,B 0,C 180,E1 -21466.577,E2 -21466.577} C_VEL
LIN {X 0,Y 208.327,Z 371.508,A -85,B 0,C 180,E1 -21470.132,E2 -21470.132} C_VEL
LIN {X 0,Y 205.183,Z 376.292,A -85,B 0,C 180,E1 -21473.169,E2 -21473.169} C_VEL
LIN {X 0,Y 202.564,Z 380.124,A -85,B 0,C 180,E1 -21476.361,E2 -21476.361} C_VEL
LIN {X 0,Y 200.002,Z 383.625,A -85,B 0,C 180,E1 -21480.528,E2 -21480.528} C_VEL
LIN {X 0,Y 198.247,Z 385.651,A -85,B 0,C 180,E1 -21484.82,E2 -21484.82} C_VEL
LIN {X 0,Y 197.283,Z 386.173,A -85,B 0,C 180,E1 -21489.128,E2 -21489.128} C_VEL
LIN {X 0,Y 196.896,Z 385.268,A -85,B 0,C 180,E1 -21493.405,E2 -21493.405} C_VEL
LIN {X 0,Y 196.941,Z 384.284,A -85,B 0,C 180,E1 -21495.531,E2 -21495.531} C_VEL
LIN {X 0,Y 197.229,Z 381.262,A -85,B 0,C 180,E1 -21499.734,E2 -21499.734} C_VEL
LIN {X 0,Y 198.011,Z 377.185,A -85,B 0,C 180,E1 -21503.539,E2 -21503.539} C_VEL
LIN {X 0,Y 198.978,Z 372.307,A -85,B 0,C 180,E1 -21506.96,E2 -21506.96} C_VEL
LIN {X 0,Y 200.494,Z 365.863,A -85,B 0,C 180,E1 -21510.499,E2 -21510.499} C_VEL
LIN {X 0,Y 202.694,Z 357.841,A -85,B 0,C 180,E1 -21513.974,E2 -21513.974} C_VEL
LIN {X 0,Y 205.051,Z 349.163,A -85,B 0,C 180,E1 -21516.986,E2 -21516.986} C_VEL
LIN {X 0,Y 207.631,Z 339.38,A -85,B 0,C 180,E1 -21519.741,E2 -21519.741} C_VEL
LIN {X 0,Y 210.102,Z 329.253,A -85,B 0,C 180,E1 -21522.065,E2 -21522.065} C_VEL
LIN {X 0,Y 212.769,Z 318.249,A -85,B 0,C 180,E1 -21524.096,E2 -21524.096} C_VEL
LIN {X 0,Y 215.28,Z 306.359,A -85,B 0,C 180,E1 -21525.864,E2 -21525.864} C_VEL
LIN {X 0,Y 217.512,Z 293.371,A -85,B 0,C 180,E1 -21527.387,E2 -21527.387} C_VEL
LIN {X 0,Y 219.461,Z 279.21,A -85,B 0,C 180,E1 -21528.614,E2 -21528.614} C_VEL
LIN {X 0,Y 220.83,Z 265.266,A -85,B 0,C 180,E1 -21529.459,E2 -21529.459} C_VEL
LIN {X 0,Y 221.883,Z 246.301,A -85,B 0,C 180,E1 -21530.146,E2 -21530.146} C_VEL
LIN {X 0,Y 225.163,Z 182.353,A -85,B 0,C 180,E1 -21532.038,E2 -21532.038} C_VEL
LIN {X 0,Y 219.585,Z 167.429,A -85,B 0,C 180,E1 -21533.543,E2 -21533.543} C_VEL
LIN {X 0,Y 213.598,Z 155.321,A -85,B 0,C 180,E1 -21535.112,E2 -21535.112} C_VEL
LIN {X 0,Y 205.427,Z 141.366,A -85,B 0,C 180,E1 -21537.344,E2 -21537.344} C_VEL
LIN {X 0,Y 201.683,Z 135.366,A -85,B 0,C 180,E1 -21538.427,E2 -21538.427} C_VEL
LIN {X 0,Y 200.034,Z 132.808,A -85,B 0,C 180,E1 -21538.917,E2 -21538.917} C_VEL
LIN {X 0,Y 199.63,Z 131.243,A -85,B 0,C 180,E1 -21539.112,E2 -21539.112} C_VEL
LIN {X 0,Y 199.635,Z 131.242,A -85,B 0,C 180,E1 -21542.354,E2 -21542.354} C_VEL
LIN {X 0,Y 199.646,Z 131.241,A -85,B 0,C 180,E1 -21546.754,E2 -21546.754} C_VEL
LIN {X 0,Y 199.696,Z 131.234,A -85,B 0,C 180,E1 -21549.303,E2 -21549.303} C_VEL
LIN {X 0,Y 199.677,Z 131.221,A -85,B 0,C 180,E1 -21552.354,E2 -21552.354} C_VEL
LIN {X 0,Y 199.667,Z 131.223,A -85,B 0,C 180,E1 -21555.265,E2 -21555.265} C_VEL
LIN {X 0,Y 199.672,Z 131.236,A -85,B 0,C 180,E1 -21558.04,E2 -21558.04} C_VEL
LIN {X 0,Y 199.677,Z 131.211,A -85,B 0,C 180,E1 -21560.739,E2 -21560.739} C_VEL
LIN {X 0,Y 199.61,Z 131.241,A -85,B 0,C 180,E1 -21565.722,E2 -21565.722} C_VEL
LIN {X 0,Y 199.673,Z 131.229,A -85,B 0,C 180,E1 -21568.141,E2 -21568.141} C_VEL
LIN {X 0,Y 199.666,Z 131.209,A -85,B 0,C 180,E1 -21572.777,E2 -21572.777} C_VEL
LIN {X 0,Y 199.74,Z 131.229,A -85,B 0,C 180,E1 -21577.237,E2 -21577.237} C_VEL
LIN {X 0,Y 199.821,Z 131.218,A -85,B 0,C 180,E1 -21581.727,E2 -21581.727} C_VEL
LIN {X 0,Y 199.835,Z 131.209,A -85,B 0,C 180,E1 -21585.756,E2 -21585.756} C_VEL
LIN {X 0,Y 200.061,Z 131.182,A -85,B 0,C 180,E1 -21589.891,E2 -21589.891} C_VEL
LIN {X 0,Y 200.026,Z 131.158,A -85,B 0,C 180,E1 -21593.956,E2 -21593.956} C_VEL
LIN {X 0,Y 200.314,Z 131.155,A -85,B 0,C 180,E1 -21597.996,E2 -21597.996} C_VEL
LIN {X 0,Y 200.473,Z 131.135,A -85,B 0,C 180,E1 -21600.007,E2 -21600.007} C_VEL
LIN {X 0,Y 200.022,Z 131.161,A -85,B 0,C 180,E1 -21604.036,E2 -21604.036} C_VEL
LIN {X 0,Y 200.105,Z 131.179,A -85,B 0,C 180,E1 -21608.082,E2 -21608.082} C_VEL
LIN {X 0,Y 199.908,Z 131.201,A -85,B 0,C 180,E1 -21612.184,E2 -21612.184} C_VEL
LIN {X 0,Y 199.801,Z 131.219,A -85,B 0,C 180,E1 -21616.35,E2 -21616.35} C_VEL
LIN {X 0,Y 199.698,Z 131.234,A -85,B 0,C 180,E1 -21620.612,E2 -21620.612} C_VEL
LIN {X 0,Y 199.672,Z 131.236,A -85,B 0,C 180,E1 -21624.991,E2 -21624.991} C_VEL
LIN {X 0,Y 199.671,Z 131.233,A -85,B 0,C 180,E1 -21629.529,E2 -21629.529} C_VEL
LIN {X 0,Y 199.673,Z 131.228,A -85,B 0,C 180,E1 -21632.362,E2 -21632.362} C_VEL
LIN {X 0,Y 199.623,Z 131.243,A -85,B 0,C 180,E1 -21636.77,E2 -21636.77} C_VEL
LIN {X 0,Y 199.602,Z 131.236,A -85,B 0,C 180,E1 -21639.336,E2 -21639.336} C_VEL
LIN {X 0,Y 199.616,Z 131.365,A -85,B 0,C 180,E1 -21643.769,E2 -21643.769} C_VEL
LIN {X 0,Y 200.24,Z 133.336,A -85,B 0,C 180,E1 -21644.788,E2 -21644.788} C_VEL
LIN {X 0,Y 202.441,Z 137.561,A -85,B 0,C 180,E1 -21645.475,E2 -21645.475} C_VEL
LIN {X 0,Y 209.739,Z 151.659,A -85,B 0,C 180,E1 -21647.616,E2 -21647.616} C_VEL
LIN {X 0,Y 212.609,Z 157.638,A -85,B 0,C 180,E1 -21648.422,E2 -21648.422} C_VEL
LIN {X 0,Y 214.651,Z 162.717,A -85,B 0,C 180,E1 -21649.012,E2 -21649.012} C_VEL
LIN {X 0,Y 215.926,Z 168.245,A -85,B 0,C 180,E1 -21649.469,E2 -21649.469} C_VEL
LIN {X 0,Y 217.099,Z 179.934,A -85,B 0,C 180,E1 -21650.146,E2 -21650.146} C_VEL
LIN {X 0,Y 217.661,Z 187.833,A -85,B 0,C 180,E1 -21650.557,E2 -21650.557} C_VEL
LIN {X 0,Y 218.586,Z 196.845,A -85,B 0,C 180,E1 -21651.068,E2 -21651.068} C_VEL
LIN {X 0,Y 214.845,Z 271.678,A -85,B 0,C 180,E1 -21653.422,E2 -21653.422} C_VEL
LIN {X 0,Y 213.356,Z 286.345,A -85,B 0,C 180,E1 -21654.223,E2 -21654.223} C_VEL
LIN {X 0,Y 211.588,Z 298.668,A -85,B 0,C 180,E1 -21655.191,E2 -21655.191} C_VEL
LIN {X 0,Y 209.149,Z 312.102,A -85,B 0,C 180,E1 -21656.62,E2 -21656.62} C_VEL
LIN {X 0,Y 206.517,Z 324.493,A -85,B 0,C 180,E1 -21658.345,E2 -21658.345} C_VEL
LIN {X 0,Y 203.772,Z 335.598,A -85,B 0,C 180,E1 -21660.282,E2 -21660.282} C_VEL
LIN {X 0,Y 201.3,Z 345.589,A -85,B 0,C 180,E1 -21662.448,E2 -21662.448} C_VEL
LIN {X 0,Y 198.605,Z 354.899,A -85,B 0,C 180,E1 -21664.875,E2 -21664.875} C_VEL
LIN {X 0,Y 196.009,Z 364.23,A -85,B 0,C 180,E1 -21667.887,E2 -21667.887} C_VEL
LIN {X 0,Y 193.926,Z 371.983,A -85,B 0,C 180,E1 -21670.967,E2 -21670.967} C_VEL
LIN {X 0,Y 192.414,Z 378.436,A -85,B 0,C 180,E1 -21674.104,E2 -21674.104} C_VEL
LIN {X 0,Y 191.193,Z 383.699,A -85,B 0,C 180,E1 -21677.262,E2 -21677.262} C_VEL
LIN {X 0,Y 190.55,Z 387.98,A -85,B 0,C 180,E1 -21680.449,E2 -21680.449} C_VEL
LIN {X 0,Y 190.233,Z 391.371,A -85,B 0,C 180,E1 -21683.64,E2 -21683.64} C_VEL
LIN {X 0,Y 190.173,Z 393.479,A -85,B 0,C 180,E1 -21686.279,E2 -21686.279} C_VEL
LIN {X 0,Y 190.307,Z 395.557,A -85,B 0,C 180,E1 -21690.003,E2 -21690.003} C_VEL
LIN {X 0,Y 190.177,Z 396.598,A -85,B 0,C 180,E1 -21694.242,E2 -21694.242} C_VEL
LIN {X 0,Y 190.472,Z 396.32,A -85,B 0,C 180,E1 -21698.49,E2 -21698.49} C_VEL
LIN {X 0,Y 191.495,Z 394.741,A -85,B 0,C 180,E1 -21702.724,E2 -21702.724} C_VEL
LIN {X 0,Y 193.456,Z 391.835,A -85,B 0,C 180,E1 -21706.899,E2 -21706.899} C_VEL
LIN {X 0,Y 196.35,Z 387.528,A -85,B 0,C 180,E1 -21710.976,E2 -21710.976} C_VEL
LIN {X 0,Y 200.084,Z 381.703,A -85,B 0,C 180,E1 -21714.932,E2 -21714.932} C_VEL
LIN {X 0,Y 204.241,Z 375.182,A -85,B 0,C 180,E1 -21718.241,E2 -21718.241} C_VEL
LIN {X 0,Y 209.079,Z 367.136,A -85,B 0,C 180,E1 -21721.404,E2 -21721.404} C_VEL
LIN {X 0,Y 213.857,Z 358.737,A -85,B 0,C 180,E1 -21723.967,E2 -21723.967} C_VEL
LIN {X 0,Y 218.697,Z 348.943,A -85,B 0,C 180,E1 -21726.397,E2 -21726.397} C_VEL
LIN {X 0,Y 223.471,Z 338.567,A -85,B 0,C 180,E1 -21728.401,E2 -21728.401} C_VEL
LIN {X 0,Y 227.858,Z 327.663,A -85,B 0,C 180,E1 -21730.083,E2 -21730.083} C_VEL
LIN {X 0,Y 231.862,Z 315.907,A -85,B 0,C 180,E1 -21731.536,E2 -21731.536} C_VEL
LIN {X 0,Y 235.663,Z 303.021,A -85,B 0,C 180,E1 -21732.726,E2 -21732.726} C_VEL
LIN {X 0,Y 238.78,Z 289.116,A -85,B 0,C 180,E1 -21733.693,E2 -21733.693} C_VEL
LIN {X 0,Y 241.046,Z 275.527,A -85,B 0,C 180,E1 -21734.337,E2 -21734.337} C_VEL
LIN {X 0,Y 242.407,Z 260.435,A -85,B 0,C 180,E1 -21734.84,E2 -21734.84} C_VEL
LIN {X 0,Y 245.667,Z 212.942,A -85,B 0,C 180,E1 -21736.125,E2 -21736.125} C_VEL
LIN {X 0,Y 241.782,Z 203.782,A -85,B 0,C 180,E1 -21737.795,E2 -21737.795} C_VEL
LIN {X 0,Y 236.983,Z 193.84,A -85,B 0,C 180,E1 -21739.971,E2 -21739.971} C_VEL
LIN {X 0,Y 231.496,Z 183.58,A -85,B 0,C 180,E1 -21742.705,E2 -21742.705} C_VEL
LIN {X 0,Y 227.997,Z 177.682,A -85,B 0,C 180,E1 -21744.604,E2 -21744.604} C_VEL
LIN {X 0,Y 225.117,Z 173.004,A -85,B 0,C 180,E1 -21746.292,E2 -21746.292} C_VEL
LIN {X 0,Y 222.163,Z 168.347,A -85,B 0,C 180,E1 -21748.171,E2 -21748.171} C_VEL
LIN {X 0,Y 218.628,Z 162.992,A -85,B 0,C 180,E1 -21750.697,E2 -21750.697} C_VEL
LIN {X 0,Y 215.473,Z 158.543,A -85,B 0,C 180,E1 -21753.283,E2 -21753.283} C_VEL
LIN {X 0,Y 214.615,Z 157.254,A -85,B 0,C 180,E1 -21754.067,E2 -21754.067} C_VEL
LIN {X 0,Y 211.872,Z 154.069,A -85,B 0,C 180,E1 -21756.757,E2 -21756.757} C_VEL
LIN {X 0,Y 209.99,Z 151.103,A -85,B 0,C 180,E1 -21759.058,E2 -21759.058} C_VEL
LIN {X 0,Y 209.151,Z 150.03,A -85,B 0,C 180,E1 -21760.205,E2 -21760.205} C_VEL
LIN {X 0,Y 205.811,Z 146.897,A -85,B 0,C 180,E1 -21766.668,E2 -21766.668} C_VEL
LIN {X 0,Y 205.232,Z 144.554,A -85,B 0,C 180,E1 -21770.135,E2 -21770.135} C_VEL
LIN {X 0,Y 205.243,Z 144.518,A -85,B 0,C 180,E1 -21774.344,E2 -21774.344} C_VEL
LIN {X 0,Y 206.522,Z 147.11,A -85,B 0,C 180,E1 -21779.506,E2 -21779.506} C_VEL
LIN {X 0,Y 208.549,Z 149.578,A -85,B 0,C 180,E1 -21783.374,E2 -21783.374} C_VEL
LIN {X 0,Y 210.089,Z 150.529,A -85,B 0,C 180,E1 -21785.392,E2 -21785.392} C_VEL
LIN {X 0,Y 211.876,Z 153.669,A -85,B 0,C 180,E1 -21787.618,E2 -21787.618} C_VEL
LIN {X 0,Y 214.35,Z 156.009,A -85,B 0,C 180,E1 -21790.012,E2 -21790.012} C_VEL
LIN {X 0,Y 216.618,Z 159.434,A -85,B 0,C 180,E1 -21792.049,E2 -21792.049} C_VEL
LIN {X 0,Y 218.484,Z 161.302,A -85,B 0,C 180,E1 -21793.479,E2 -21793.479} C_VEL
LIN {X 0,Y 221.18,Z 165.047,A -85,B 0,C 180,E1 -21795.449,E2 -21795.449} C_VEL
LIN {X 0,Y 223.005,Z 167.546,A -85,B 0,C 180,E1 -21796.647,E2 -21796.647} C_VEL
LIN {X 0,Y 226.054,Z 171.566,A -85,B 0,C 180,E1 -21798.491,E2 -21798.491} C_VEL
LIN {X 0,Y 229.516,Z 176.419,A -85,B 0,C 180,E1 -21800.419,E2 -21800.419} C_VEL
LIN {X 0,Y 234.641,Z 184.088,A -85,B 0,C 180,E1 -21803.014,E2 -21803.014} C_VEL
LIN {X 0,Y 240.552,Z 194.699,A -85,B 0,C 180,E1 -21805.752,E2 -21805.752} C_VEL
LIN {X 0,Y 246.022,Z 206.06,A -85,B 0,C 180,E1 -21808.073,E2 -21808.073} C_VEL
LIN {X 0,Y 244.94,Z 223.312,A -85,B 0,C 180,E1 -21808.572,E2 -21808.572} C_VEL
LIN {X 0,Y 242.012,Z 263.117,A -85,B 0,C 180,E1 -21809.68,E2 -21809.68} C_VEL
LIN {X 0,Y 240.036,Z 277.163,A -85,B 0,C 180,E1 -21810.32,E2 -21810.32} C_VEL
LIN {X 0,Y 237.272,Z 290.68,A -85,B 0,C 180,E1 -21811.205,E2 -21811.205} C_VEL
LIN {X 0,Y 234.058,Z 303.413,A -85,B 0,C 180,E1 -21812.377,E2 -21812.377} C_VEL
LIN {X 0,Y 230.13,Z 315.836,A -85,B 0,C 180,E1 -21813.845,E2 -21813.845} C_VEL
LIN {X 0,Y 225.731,Z 327.393,A -85,B 0,C 180,E1 -21815.568,E2 -21815.568} C_VEL
LIN {X 0,Y 220.879,Z 338.489,A -85,B 0,C 180,E1 -21817.672,E2 -21817.672} C_VEL
LIN {X 0,Y 215.917,Z 348.552,A -85,B 0,C 180,E1 -21820.099,E2 -21820.099} C_VEL
LIN {X 0,Y 210.957,Z 357.585,A -85,B 0,C 180,E1 -21822.864,E2 -21822.864} C_VEL
LIN {X 0,Y 206.796,Z 364.469,A -85,B 0,C 180,E1 -21825.525,E2 -21825.525} C_VEL
LIN {X 0,Y 202.56,Z 371.066,A -85,B 0,C 180,E1 -21828.756,E2 -21828.756} C_VEL
LIN {X 0,Y 199.138,Z 375.971,A -85,B 0,C 180,E1 -21831.855,E2 -21831.855} C_VEL
LIN {X 0,Y 195.936,Z 380.386,A -85,B 0,C 180,E1 -21835.572,E2 -21835.572} C_VEL
LIN {X 0,Y 193.41,Z 383.559,A -85,B 0,C 180,E1 -21839.418,E2 -21839.418} C_VEL
LIN {X 0,Y 191.427,Z 385.717,A -85,B 0,C 180,E1 -21843.857,E2 -21843.857} C_VEL
LIN {X 0,Y 190.309,Z 386.4,A -85,B 0,C 180,E1 -21848.325,E2 -21848.325} C_VEL
LIN {X 0,Y 189.822,Z 385.617,A -85,B 0,C 180,E1 -21852.768,E2 -21852.768} C_VEL
LIN {X 0,Y 189.838,Z 384.691,A -85,B 0,C 180,E1 -21854.978,E2 -21854.978} C_VEL
LIN {X 0,Y 190.087,Z 381.783,A -85,B 0,C 180,E1 -21859.344,E2 -21859.344} C_VEL
LIN {X 0,Y 190.915,Z 377.464,A -85,B 0,C 180,E1 -21863.603,E2 -21863.603} C_VEL
LIN {X 0,Y 191.814,Z 373.078,A -85,B 0,C 180,E1 -21866.847,E2 -21866.847} C_VEL
LIN {X 0,Y 193.342,Z 366.775,A -85,B 0,C 180,E1 -21870.518,E2 -21870.518} C_VEL
LIN {X 0,Y 195.559,Z 358.912,A -85,B 0,C 180,E1 -21874.119,E2 -21874.119} C_VEL
LIN {X 0,Y 197.989,Z 350.408,A -85,B 0,C 180,E1 -21877.236,E2 -21877.236} C_VEL
LIN {X 0,Y 200.656,Z 340.827,A -85,B 0,C 180,E1 -21880.083,E2 -21880.083} C_VEL
LIN {X 0,Y 203.116,Z 330.967,A -85,B 0,C 180,E1 -21882.486,E2 -21882.486} C_VEL
LIN {X 0,Y 206.192,Z 318.971,A -85,B 0,C 180,E1 -21884.808,E2 -21884.808} C_VEL
LIN {X 0,Y 208.771,Z 307.205,A -85,B 0,C 180,E1 -21886.624,E2 -21886.624} C_VEL
LIN {X 0,Y 211.125,Z 294.389,A -85,B 0,C 180,E1 -21888.182,E2 -21888.182} C_VEL
LIN {X 0,Y 213.043,Z 281.32,A -85,B 0,C 180,E1 -21889.384,E2 -21889.384} C_VEL
LIN {X 0,Y 214.492,Z 267.345,A -85,B 0,C 180,E1 -21890.308,E2 -21890.308} C_VEL
LIN {X 0,Y 215.586,Z 251.032,A -85,B 0,C 180,E1 -21890.948,E2 -21890.948} C_VEL
LIN {X 0,Y 219.115,Z 184.231,A -85,B 0,C 180,E1 -21892.967,E2 -21892.967} C_VEL
LIN {X 0,Y 214.539,Z 171.644,A -85,B 0,C 180,E1 -21894.272,E2 -21894.272} C_VEL
LIN {X 0,Y 209.842,Z 161.855,A -85,B 0,C 180,E1 -21895.563,E2 -21895.563} C_VEL
LIN {X 0,Y 201.776,Z 147.456,A -85,B 0,C 180,E1 -21897.862,E2 -21897.862} C_VEL
LIN {X 0,Y 197.025,Z 140.007,A -85,B 0,C 180,E1 -21899.282,E2 -21899.282} C_VEL
LIN {X 0,Y 194.582,Z 136.214,A -85,B 0,C 180,E1 -21900.049,E2 -21900.049} C_VEL
LIN {X 0,Y 193.065,Z 133.935,A -85,B 0,C 180,E1 -21900.536,E2 -21900.536} C_VEL
LIN {X 0,Y 192.575,Z 132.12,A -85,B 0,C 180,E1 -21900.791,E2 -21900.791} C_VEL
LIN {X 0,Y 192.592,Z 132.117,A -85,B 0,C 180,E1 -21905.719,E2 -21905.719} C_VEL
LIN {X 0,Y 192.605,Z 132.118,A -85,B 0,C 180,E1 -21909.993,E2 -21909.993} C_VEL
LIN {X 0,Y 192.604,Z 132.093,A -85,B 0,C 180,E1 -21913.887,E2 -21913.887} C_VEL
LIN {X 0,Y 192.584,Z 132.113,A -85,B 0,C 180,E1 -21918.949,E2 -21918.949} C_VEL
LIN {X 0,Y 192.595,Z 132.096,A -85,B 0,C 180,E1 -21923.393,E2 -21923.393} C_VEL
LIN {X 0,Y 192.582,Z 132.117,A -85,B 0,C 180,E1 -21927.066,E2 -21927.066} C_VEL
LIN {X 0,Y 192.639,Z 132.077,A -85,B 0,C 180,E1 -21931.697,E2 -21931.697} C_VEL
LIN {X 0,Y 192.697,Z 132.108,A -85,B 0,C 180,E1 -21936.356,E2 -21936.356} C_VEL
LIN {X 0,Y 192.765,Z 132.095,A -85,B 0,C 180,E1 -21941.419,E2 -21941.419} C_VEL
LIN {X 0,Y 192.839,Z 132.086,A -85,B 0,C 180,E1 -21947.377,E2 -21947.377} C_VEL
LIN {X 0,Y 193.059,Z 132.038,A -85,B 0,C 180,E1 -21951.634,E2 -21951.634} C_VEL
LIN {X 0,Y 193.256,Z 132.033,A -85,B 0,C 180,E1 -21957.923,E2 -21957.923} C_VEL
LIN {X 0,Y 193.437,Z 132.011,A -85,B 0,C 180,E1 -21960.007,E2 -21960.007} C_VEL
LIN {X 0,Y 192.968,Z 132.038,A -85,B 0,C 180,E1 -21964.184,E2 -21964.184} C_VEL
LIN {X 0,Y 193.056,Z 132.057,A -85,B 0,C 180,E1 -21968.38,E2 -21968.38} C_VEL
LIN {X 0,Y 192.848,Z 132.081,A -85,B 0,C 180,E1 -21972.637,E2 -21972.637} C_VEL
LIN {X 0,Y 192.754,Z 132.094,A -85,B 0,C 180,E1 -21976.966,E2 -21976.966} C_VEL
LIN {X 0,Y 192.634,Z 132.113,A -85,B 0,C 180,E1 -21981.404,E2 -21981.404} C_VEL
LIN {X 0,Y 192.663,Z 132.108,A -85,B 0,C 180,E1 -21984.231,E2 -21984.231} C_VEL
LIN {X 0,Y 192.649,Z 132.104,A -85,B 0,C 180,E1 -21988.898,E2 -21988.898} C_VEL
LIN {X 0,Y 192.599,Z 132.112,A -85,B 0,C 180,E1 -21993.193,E2 -21993.193} C_VEL
LIN {X 0,Y 192.548,Z 132.124,A -85,B 0,C 180,E1 -21998.36,E2 -21998.36} C_VEL
LIN {X 0,Y 192.568,Z 132.307,A -85,B 0,C 180,E1 -22002.582,E2 -22002.582} C_VEL
LIN {X 0,Y 192.802,Z 133.309,A -85,B 0,C 180,E1 -22002.991,E2 -22002.991} C_VEL
LIN {X 0,Y 194.704,Z 136.744,A -85,B 0,C 180,E1 -22003.633,E2 -22003.633} C_VEL
LIN {X 0,Y 196.522,Z 139.895,A -85,B 0,C 180,E1 -22004.223,E2 -22004.223} C_VEL
LIN {X 0,Y 202.933,Z 151.939,A -85,B 0,C 180,E1 -22006.225,E2 -22006.225} C_VEL
LIN {X 0,Y 209.292,Z 165.693,A -85,B 0,C 180,E1 -22008.119,E2 -22008.119} C_VEL
LIN {X 0,Y 216.439,Z 184.069,A -85,B 0,C 180,E1 -22010.194,E2 -22010.194} C_VEL
LIN {X 0,Y 217.661,Z 187.833,A -85,B 0,C 180,E1 -22010.557,E2 -22010.557} C_VEL
LIN {X 0,Y 217.381,Z 191.741,A -85,B 0,C 180,E1 -22010.662,E2 -22010.662} C_VEL
LIN {X 0,Y 215.218,Z 198.061,A -85,B 0,C 180,E1 -22010.537,E2 -22010.537} C_VEL
LIN {X 0,Y 212.775,Z 204.404,A -85,B 0,C 180,E1 -22010.361,E2 -22010.361} C_VEL
LIN {X 0,Y 212.083,Z 208.38,A -85,B 0,C 180,E1 -22010.399,E2 -22010.399} C_VEL
LIN {X 0,Y 208.768,Z 271.553,A -85,B 0,C 180,E1 -22012.437,E2 -22012.437} C_VEL
LIN {X 0,Y 207.258,Z 285.844,A -85,B 0,C 180,E1 -22013.226,E2 -22013.226} C_VEL
LIN {X 0,Y 205.342,Z 298.826,A -85,B 0,C 180,E1 -22014.273,E2 -22014.273} C_VEL
LIN {X 0,Y 202.819,Z 312.187,A -85,B 0,C 180,E1 -22015.734,E2 -22015.734} C_VEL
LIN {X 0,Y 200.041,Z 324.756,A -85,B 0,C 180,E1 -22017.54,E2 -22017.54} C_VEL
LIN {X 0,Y 197.251,Z 335.597,A -85,B 0,C 180,E1 -22019.491,E2 -22019.491} C_VEL
LIN {X 0,Y 194.356,Z 346.546,A -85,B 0,C 180,E1 -22021.964,E2 -22021.964} C_VEL
LIN {X 0,Y 191.612,Z 355.668,A -85,B 0,C 180,E1 -22024.474,E2 -22024.474} C_VEL
LIN {X 0,Y 188.958,Z 364.838,A -85,B 0,C 180,E1 -22027.593,E2 -22027.593} C_VEL
LIN {X 0,Y 186.856,Z 372.453,A -85,B 0,C 180,E1 -22030.789,E2 -22030.789} C_VEL
LIN {X 0,Y 185.041,Z 379.704,A -85,B 0,C 180,E1 -22034.585,E2 -22034.585} C_VEL
LIN {X 0,Y 183.933,Z 384.736,A -85,B 0,C 180,E1 -22037.872,E2 -22037.872} C_VEL
LIN {X 0,Y 183.251,Z 389.901,A -85,B 0,C 180,E1 -22042.289,E2 -22042.289} C_VEL
LIN {X 0,Y 183.09,Z 393.36,A -85,B 0,C 180,E1 -22046.481,E2 -22046.481} C_VEL
LIN {X 0,Y 183.211,Z 395.277,A -85,B 0,C 180,E1 -22050.003,E2 -22050.003} C_VEL
LIN {X 0,Y 183.09,Z 396.385,A -85,B 0,C 180,E1 -22054.406,E2 -22054.406} C_VEL
LIN {X 0,Y 183.422,Z 396.173,A -85,B 0,C 180,E1 -22058.819,E2 -22058.819} C_VEL
LIN {X 0,Y 184.52,Z 394.663,A -85,B 0,C 180,E1 -22063.214,E2 -22063.214} C_VEL
LIN {X 0,Y 186.641,Z 391.832,A -85,B 0,C 180,E1 -22067.535,E2 -22067.535} C_VEL
LIN {X 0,Y 189.684,Z 387.602,A -85,B 0,C 180,E1 -22071.75,E2 -22071.75} C_VEL
LIN {X 0,Y 193.642,Z 381.856,A -85,B 0,C 180,E1 -22075.822,E2 -22075.822} C_VEL
LIN {X 0,Y 198.011,Z 375.421,A -85,B 0,C 180,E1 -22079.214,E2 -22079.214} C_VEL
LIN {X 0,Y 203.06,Z 367.472,A -85,B 0,C 180,E1 -22082.446,E2 -22082.446} C_VEL
LIN {X 0,Y 208.028,Z 359.181,A -85,B 0,C 180,E1 -22085.056,E2 -22085.056} C_VEL
LIN {X 0,Y 213.431,Z 348.79,A -85,B 0,C 180,E1 -22087.694,E2 -22087.694} C_VEL
LIN {X 0,Y 218.497,Z 338.247,A -85,B 0,C 180,E1 -22089.741,E2 -22089.741} C_VEL
LIN {X 0,Y 223.531,Z 325.963,A -85,B 0,C 180,E1 -22091.623,E2 -22091.623} C_VEL
LIN {X 0,Y 227.746,Z 313.849,A -85,B 0,C 180,E1 -22093.062,E2 -22093.062} C_VEL
LIN {X 0,Y 231.65,Z 300.404,A -85,B 0,C 180,E1 -22094.253,E2 -22094.253} C_VEL
LIN {X 0,Y 234.793,Z 286.368,A -85,B 0,C 180,E1 -22095.159,E2 -22095.159} C_VEL
LIN {X 0,Y 236.949,Z 272.384,A -85,B 0,C 180,E1 -22095.791,E2 -22095.791} C_VEL
LIN {X 0,Y 239.084,Z 245.223,A -85,B 0,C 180,E1 -22096.585,E2 -22096.585} C_VEL
LIN {X 0,Y 241.194,Z 215.547,A -85,B 0,C 180,E1 -22097.393,E2 -22097.393} C_VEL
LIN {X 0,Y 236.773,Z 205.194,A -85,B 0,C 180,E1 -22099.427,E2 -22099.427} C_VEL
LIN {X 0,Y 231.147,Z 193.693,A -85,B 0,C 180,E1 -22102.238,E2 -22102.238} C_VEL
LIN {X 0,Y 225.852,Z 184.137,A -85,B 0,C 180,E1 -22105.172,E2 -22105.172} C_VEL
LIN {X 0,Y 222.148,Z 177.974,A -85,B 0,C 180,E1 -22107.459,E2 -22107.459} C_VEL
LIN {X 0,Y 219.591,Z 173.887,A -85,B 0,C 180,E1 -22109.192,E2 -22109.192} C_VEL
LIN {X 0,Y 216.559,Z 169.139,A -85,B 0,C 180,E1 -22111.516,E2 -22111.516} C_VEL
LIN {X 0,Y 213.666,Z 164.807,A -85,B 0,C 180,E1 -22114.034,E2 -22114.034} C_VEL
LIN {X 0,Y 210.847,Z 161.166,A -85,B 0,C 180,E1 -22116.857,E2 -22116.857} C_VEL
LIN {X 0,Y 208.755,Z 158.083,A -85,B 0,C 180,E1 -22119.437,E2 -22119.437} C_VEL
LIN {X 0,Y 208.195,Z 157.08,A -85,B 0,C 180,E1 -22120.265,E2 -22120.265} C_VEL
LIN {X 0,Y 204.8,Z 153.762,A -85,B 0,C 180,E1 -22127.105,E2 -22127.105} C_VEL
LIN {X 0,Y 204.297,Z 151.513,A -85,B 0,C 180,E1 -22130.647,E2 -22130.647} C_VEL
LIN {X 0,Y 204.35,Z 151.619,A -85,B 0,C 180,E1 -22134.319,E2 -22134.319} C_VEL
LIN {X 0,Y 205.576,Z 154.176,A -85,B 0,C 180,E1 -22139.381,E2 -22139.381} C_VEL
LIN {X 0,Y 207.663,Z 156.641,A -85,B 0,C 180,E1 -22143.389,E2 -22143.389} C_VEL
LIN {X 0,Y 208.806,Z 157.398,A -85,B 0,C 180,E1 -22144.941,E2 -22144.941} C_VEL
LIN {X 0,Y 210.566,Z 160.485,A -85,B 0,C 180,E1 -22147.209,E2 -22147.209} C_VEL
LIN {X 0,Y 212.832,Z 162.77,A -85,B 0,C 180,E1 -22149.497,E2 -22149.497} C_VEL
LIN {X 0,Y 215.241,Z 166.295,A -85,B 0,C 180,E1 -22151.717,E2 -22151.717} C_VEL
LIN {X 0,Y 216.785,Z 168.006,A -85,B 0,C 180,E1 -22152.953,E2 -22152.953} C_VEL
LIN {X 0,Y 219.641,Z 171.863,A -85,B 0,C 180,E1 -22155.092,E2 -22155.092} C_VEL
LIN {X 0,Y 224.025,Z 178.084,A -85,B 0,C 180,E1 -22157.941,E2 -22157.941} C_VEL
LIN {X 0,Y 227.365,Z 182.914,A -85,B 0,C 180,E1 -22159.871,E2 -22159.871} C_VEL
LIN {X 0,Y 232.368,Z 190.603,A -85,B 0,C 180,E1 -22162.493,E2 -22162.493} C_VEL
LIN {X 0,Y 237.956,Z 201.284,A -85,B 0,C 180,E1 -22165.204,E2 -22165.204} C_VEL
LIN {X 0,Y 241.621,Z 209.107,A -85,B 0,C 180,E1 -22166.842,E2 -22166.842} C_VEL
LIN {X 0,Y 237.619,Z 263.021,A -85,B 0,C 180,E1 -22168.343,E2 -22168.343} C_VEL
LIN {X 0,Y 235.541,Z 277.384,A -85,B 0,C 180,E1 -22168.997,E2 -22168.997} C_VEL
LIN {X 0,Y 232.613,Z 291.254,A -85,B 0,C 180,E1 -22169.913,E2 -22169.913} C_VEL
LIN {X 0,Y 229.25,Z 303.999,A -85,B 0,C 180,E1 -22171.097,E2 -22171.097} C_VEL
LIN {X 0,Y 225.186,Z 316.356,A -85,B 0,C 180,E1 -22172.574,E2 -22172.574} C_VEL
LIN {X 0,Y 220.443,Z 328.294,A -85,B 0,C 180,E1 -22174.383,E2 -22174.383} C_VEL
LIN {X 0,Y 215.362,Z 339.335,A -85,B 0,C 180,E1 -22176.521,E2 -22176.521} C_VEL
LIN {X 0,Y 210.21,Z 349.27,A -85,B 0,C 180,E1 -22178.98,E2 -22178.98} C_VEL
LIN {X 0,Y 205.033,Z 358.188,A -85,B 0,C 180,E1 -22181.791,E2 -22181.791} C_VEL
LIN {X 0,Y 200.857,Z 364.769,A -85,B 0,C 180,E1 -22184.4,E2 -22184.4} C_VEL
LIN {X 0,Y 196.895,Z 370.604,A -85,B 0,C 180,E1 -22187.294,E2 -22187.294} C_VEL
LIN {X 0,Y 193.218,Z 375.652,A -85,B 0,C 180,E1 -22190.463,E2 -22190.463} C_VEL
LIN {X 0,Y 189.314,Z 380.671,A -85,B 0,C 180,E1 -22194.743,E2 -22194.743} C_VEL
LIN {X 0,Y 186.923,Z 383.499,A -85,B 0,C 180,E1 -22198.236,E2 -22198.236} C_VEL
LIN {X 0,Y 184.676,Z 385.776,A -85,B 0,C 180,E1 -22202.824,E2 -22202.824} C_VEL
LIN {X 0,Y 183.382,Z 386.581,A -85,B 0,C 180,E1 -22207.462,E2 -22207.462} C_VEL
LIN {X 0,Y 182.757,Z 385.953,A -85,B 0,C 180,E1 -22212.08,E2 -22212.08} C_VEL
LIN {X 0,Y 182.729,Z 385.096,A -85,B 0,C 180,E1 -22214.378,E2 -22214.378} C_VEL
LIN {X 0,Y 182.922,Z 382.306,A -85,B 0,C 180,E1 -22218.921,E2 -22218.921} C_VEL
LIN {X 0,Y 183.509,Z 379.268,A -85,B 0,C 180,E1 -22222.294,E2 -22222.294} C_VEL
LIN {X 0,Y 184.329,Z 375.333,A -85,B 0,C 180,E1 -22225.624,E2 -22225.624} C_VEL
LIN {X 0,Y 185.467,Z 370.487,A -85,B 0,C 180,E1 -22228.911,E2 -22228.911} C_VEL
LIN {X 0,Y 187.399,Z 363.476,A -85,B 0,C 180,E1 -22232.684,E2 -22232.684} C_VEL
LIN {X 0,Y 189.979,Z 354.786,A -85,B 0,C 180,E1 -22236.369,E2 -22236.369} C_VEL
LIN {X 0,Y 192.502,Z 346.275,A -85,B 0,C 180,E1 -22239.268,E2 -22239.268} C_VEL
LIN {X 0,Y 195.087,Z 336.709,A -85,B 0,C 180,E1 -22241.952,E2 -22241.952} C_VEL
LIN {X 0,Y 198.075,Z 325.916,A -85,B 0,C 180,E1 -22244.378,E2 -22244.378} C_VEL
LIN {X 0,Y 200.942,Z 314.142,A -85,B 0,C 180,E1 -22246.506,E2 -22246.506} C_VEL
LIN {X 0,Y 203.661,Z 301.182,A -85,B 0,C 180,E1 -22248.351,E2 -22248.351} C_VEL
LIN {X 0,Y 206.044,Z 287.644,A -85,B 0,C 180,E1 -22249.81,E2 -22249.81} C_VEL
LIN {X 0,Y 207.79,Z 273.54,A -85,B 0,C 180,E1 -22250.928,E2 -22250.928} C_VEL
LIN {X 0,Y 209.031,Z 259.912,A -85,B 0,C 180,E1 -22251.638,E2 -22251.638} C_VEL
LIN {X 0,Y 213.003,Z 185.472,A -85,B 0,C 180,E1 -22253.992,E2 -22253.992} C_VEL
LIN {X 0,Y 208.337,Z 172.93,A -85,B 0,C 180,E1 -22255.391,E2 -22255.391} C_VEL
LIN {X 0,Y 201.428,Z 159.522,A -85,B 0,C 180,E1 -22257.397,E2 -22257.397} C_VEL
LIN {X 0,Y 194.601,Z 147.907,A -85,B 0,C 180,E1 -22259.486,E2 -22259.486} C_VEL
LIN {X 0,Y 190.208,Z 141.127,A -85,B 0,C 180,E1 -22260.911,E2 -22260.911} C_VEL
LIN {X 0,Y 187.738,Z 137.263,A -85,B 0,C 180,E1 -22261.758,E2 -22261.758} C_VEL
LIN {X 0,Y 186.027,Z 134.816,A -85,B 0,C 180,E1 -22262.353,E2 -22262.353} C_VEL
LIN {X 0,Y 185.558,Z 132.994,A -85,B 0,C 180,E1 -22262.662,E2 -22262.662} C_VEL
LIN {X 0,Y 185.569,Z 132.995,A -85,B 0,C 180,E1 -22267.328,E2 -22267.328} C_VEL
LIN {X 0,Y 185.569,Z 132.993,A -85,B 0,C 180,E1 -22270.773,E2 -22270.773} C_VEL
LIN {X 0,Y 185.561,Z 132.987,A -85,B 0,C 180,E1 -22276.018,E2 -22276.018} C_VEL
LIN {X 0,Y 185.541,Z 132.977,A -85,B 0,C 180,E1 -22279.925,E2 -22279.925} C_VEL
LIN {X 0,Y 185.551,Z 132.966,A -85,B 0,C 180,E1 -22282.708,E2 -22282.708} C_VEL
LIN {X 0,Y 185.518,Z 132.993,A -85,B 0,C 180,E1 -22287.98,E2 -22287.98} C_VEL
LIN {X 0,Y 185.559,Z 132.96,A -85,B 0,C 180,E1 -22290.582,E2 -22290.582} C_VEL
LIN {X 0,Y 185.586,Z 132.988,A -85,B 0,C 180,E1 -22295.391,E2 -22295.391} C_VEL
LIN {X 0,Y 185.694,Z 132.975,A -85,B 0,C 180,E1 -22301.106,E2 -22301.106} C_VEL
LIN {X 0,Y 185.716,Z 132.968,A -85,B 0,C 180,E1 -22304.647,E2 -22304.647} C_VEL
LIN {X 0,Y 185.929,Z 132.946,A -85,B 0,C 180,E1 -22309.335,E2 -22309.335} C_VEL
LIN {X 0,Y 185.953,Z 132.907,A -85,B 0,C 180,E1 -22313.497,E2 -22313.497} C_VEL
LIN {X 0,Y 186.2,Z 132.91,A -85,B 0,C 180,E1 -22317.844,E2 -22317.844} C_VEL
LIN {X 0,Y 186.4,Z 132.888,A -85,B 0,C 180,E1 -22320.007,E2 -22320.007} C_VEL
LIN {X 0,Y 185.915,Z 132.914,A -85,B 0,C 180,E1 -22324.343,E2 -22324.343} C_VEL
LIN {X 0,Y 186.003,Z 132.937,A -85,B 0,C 180,E1 -22328.7,E2 -22328.7} C_VEL
LIN {X 0,Y 185.759,Z 132.965,A -85,B 0,C 180,E1 -22333.128,E2 -22333.128} C_VEL
LIN {X 0,Y 185.687,Z 132.974,A -85,B 0,C 180,E1 -22337.632,E2 -22337.632} C_VEL
LIN {X 0,Y 185.595,Z 132.991,A -85,B 0,C 180,E1 -22342.258,E2 -22342.258} C_VEL
LIN {X 0,Y 185.563,Z 132.985,A -85,B 0,C 180,E1 -22347.039,E2 -22347.039} C_VEL
LIN {X 0,Y 185.579,Z 132.988,A -85,B 0,C 180,E1 -22349.5,E2 -22349.5} C_VEL
LIN {X 0,Y 185.501,Z 133.001,A -85,B 0,C 180,E1 -22354.639,E2 -22354.639} C_VEL
LIN {X 0,Y 185.505,Z 133.002,A -85,B 0,C 180,E1 -22357.321,E2 -22357.321} C_VEL
LIN {X 0,Y 185.465,Z 132.992,A -85,B 0,C 180,E1 -22361.026,E2 -22361.026} C_VEL
LIN {X 0,Y 186.537,Z 135.932,A -85,B 0,C 180,E1 -22361.475,E2 -22361.475} C_VEL
LIN {X 0,Y 188.424,Z 138.318,A -85,B 0,C 180,E1 -22362.105,E2 -22362.105} C_VEL
LIN {X 0,Y 191.861,Z 144.175,A -85,B 0,C 180,E1 -22363.284,E2 -22363.284} C_VEL
LIN {X 0,Y 198.307,Z 156.615,A -85,B 0,C 180,E1 -22365.415,E2 -22365.415} C_VEL
LIN {X 0,Y 204.22,Z 169.661,A -85,B 0,C 180,E1 -22367.274,E2 -22367.274} C_VEL
LIN {X 0,Y 211.158,Z 187.749,A -85,B 0,C 180,E1 -22369.391,E2 -22369.391} C_VEL
LIN {X 0,Y 211.888,Z 190.339,A -85,B 0,C 180,E1 -22369.631,E2 -22369.631} C_VEL
LIN {X 0,Y 212.606,Z 197.8,A -85,B 0,C 180,E1 -22370.064,E2 -22370.064} C_VEL
LIN {X 0,Y 212.083,Z 208.38,A -85,B 0,C 180,E1 -22370.399,E2 -22370.399} C_VEL
LIN {X 0,Y 211.26,Z 214.219,A -85,B 0,C 180,E1 -22370.49,E2 -22370.49} C_VEL
LIN {X 0,Y 205.405,Z 233.164,A -85,B 0,C 180,E1 -22370.215,E2 -22370.215} C_VEL
LIN {X 0,Y 204.554,Z 239.005,A -85,B 0,C 180,E1 -22370.303,E2 -22370.303} C_VEL
LIN {X 0,Y 202.633,Z 272.576,A -85,B 0,C 180,E1 -22371.453,E2 -22371.453} C_VEL
LIN {X 0,Y 201.036,Z 286.822,A -85,B 0,C 180,E1 -22372.285,E2 -22372.285} C_VEL
LIN {X 0,Y 199.15,Z 298.928,A -85,B 0,C 180,E1 -22373.297,E2 -22373.297} C_VEL
LIN {X 0,Y 196.539,Z 312.225,A -85,B 0,C 180,E1 -22374.791,E2 -22374.791} C_VEL
LIN {X 0,Y 193.843,Z 323.964,A -85,B 0,C 180,E1 -22376.51,E2 -22376.51} C_VEL
LIN {X 0,Y 191.161,Z 334.378,A -85,B 0,C 180,E1 -22378.41,E2 -22378.41} C_VEL
LIN {X 0,Y 188.099,Z 345.497,A -85,B 0,C 180,E1 -22380.944,E2 -22380.944} C_VEL
LIN {X 0,Y 185.157,Z 354.756,A -85,B 0,C 180,E1 -22383.517,E2 -22383.517} C_VEL
LIN {X 0,Y 182.349,Z 364.05,A -85,B 0,C 180,E1 -22386.735,E2 -22386.735} C_VEL
LIN {X 0,Y 179.802,Z 372.911,A -85,B 0,C 180,E1 -22390.598,E2 -22390.598} C_VEL
LIN {X 0,Y 178.145,Z 379.116,A -85,B 0,C 180,E1 -22393.973,E2 -22393.973} C_VEL
LIN {X 0,Y 176.951,Z 384.233,A -85,B 0,C 180,E1 -22397.386,E2 -22397.386} C_VEL
LIN {X 0,Y 176.18,Z 389.477,A -85,B 0,C 180,E1 -22401.978,E2 -22401.978} C_VEL
LIN {X 0,Y 176.011,Z 393.229,A -85,B 0,C 180,E1 -22406.684,E2 -22406.684} C_VEL
LIN {X 0,Y 176.116,Z 394.993,A -85,B 0,C 180,E1 -22410.003,E2 -22410.003} C_VEL
LIN {X 0,Y 175.989,Z 396.171,A -85,B 0,C 180,E1 -22414.584,E2 -22414.584} C_VEL
LIN {X 0,Y 176.369,Z 396.028,A -85,B 0,C 180,E1 -22419.175,E2 -22419.175} C_VEL
LIN {X 0,Y 177.563,Z 394.588,A -85,B 0,C 180,E1 -22423.741,E2 -22423.741} C_VEL
LIN {X 0,Y 179.855,Z 391.829,A -85,B 0,C 180,E1 -22428.22,E2 -22428.22} C_VEL
LIN {X 0,Y 183.062,Z 387.674,A -85,B 0,C 180,E1 -22432.58,E2 -22432.58} C_VEL
LIN {X 0,Y 187.268,Z 382.008,A -85,B 0,C 180,E1 -22436.769,E2 -22436.769} C_VEL
LIN {X 0,Y 192.548,Z 374.663,A -85,B 0,C 180,E1 -22440.734,E2 -22440.734} C_VEL
